// ---- DUTs/IO/PDOs/DO_X06_Pin4_Output_42CA91F7.TcDUT
{attribute 'GeneratedUsingTerminal: EP4378-1022-0017'}
{attribute addProperty BoxType "EP4378-1022-0017"}
{attribute addProperty Id "OutputAT %Q*BOOL1"}
{attribute addProperty CRC "1120571895"}
{attribute addProperty Size "1"}
TYPE DO_X06_Pin4_Output_42CA91F7 EXTENDS OutputBase_10CEE7DE :
STRUCT
	{attribute addProperty Name "Output"}
	Output AT %Q* : BOOL;
END_STRUCT
END_TYPE

// ---- DUTs/IO/PDOs/DO_X07_Pin4_Output_42CA91F7.TcDUT
{attribute 'GeneratedUsingTerminal: EP4378-1022-0017'}
{attribute addProperty BoxType "EP4378-1022-0017"}
{attribute addProperty Id "OutputAT %Q*BOOL1"}
{attribute addProperty CRC "1120571895"}
{attribute addProperty Size "1"}
TYPE DO_X07_Pin4_Output_42CA91F7 EXTENDS OutputBase_10CEE7DE :
STRUCT
	{attribute addProperty Name "Output"}
	Output AT %Q* : BOOL;
END_STRUCT
END_TYPE

// ---- DUTs/IO/PDOs/DO_X08_Pin4_Output_42CA91F7.TcDUT
{attribute 'GeneratedUsingTerminal: EP4378-1022-0017'}
{attribute addProperty BoxType "EP4378-1022-0017"}
{attribute addProperty Id "OutputAT %Q*BOOL1"}
{attribute addProperty CRC "1120571895"}
{attribute addProperty Size "1"}
TYPE DO_X08_Pin4_Output_42CA91F7 EXTENDS OutputBase_10CEE7DE :
STRUCT
	{attribute addProperty Name "Output"}
	Output AT %Q* : BOOL;
END_STRUCT
END_TYPE

// ---- DUTs/IO/PDOs/SSI_Inputs_0E3D8E33.TcDUT
{attribute 'GeneratedUsingTerminal: EP5001-0002-0016'}
{attribute addProperty BoxType "EP5001-0002-0016"}
{attribute addProperty Id "StatusAT %I*Status_ACC8459F6Counter_valueAT %I*UDINT4"}
{attribute addProperty CRC "238915123"}
{attribute addProperty Size "10"}
TYPE SSI_Inputs_0E3D8E33 EXTENDS InputBase_8311D824 :
STRUCT
	{attribute addProperty Name "Status"}
	Status AT %I* : Status_ACC8459F;
	{attribute addProperty Name "Counter_value"}
	Counter_value AT %I* : UDINT;
END_STRUCT
END_TYPE

// ---- DUTs/IO/PDOs/ENC_Status_compact_F4F89583.TcDUT
{attribute 'GeneratedUsingTerminal: EP5101-0002-0016'}
{attribute addProperty BoxType "EP5101-0002-0016"}
{attribute addProperty Id "StatusAT %I*Status_3A9E406C12Counter_valueAT %I*UINT2Latch_valueAT %I*UINT2"}
{attribute addProperty CRC "4109931907"}
{attribute addProperty Size "16"}
TYPE ENC_Status_compact_F4F89583 EXTENDS InputBase_8311D824 :
STRUCT
	{attribute addProperty Name "Status"}
	Status AT %I* : Status_3A9E406C;
	{attribute addProperty Name "Counter_value"}
	Counter_value AT %I* : UINT;
	{attribute addProperty Name "Latch_value"}
	Latch_value AT %I* : UINT;
END_STRUCT
END_TYPE

// ---- DUTs/IO/PDOs/ENC_Control_compact_E6DC9B25.TcDUT
{attribute 'GeneratedUsingTerminal: EP5101-0002-0016'}
{attribute addProperty BoxType "EP5101-0002-0016"}
{attribute addProperty Id "ControlAT %Q*Control_D500AB792Set_counter_valueAT %Q*UINT2"}
{attribute addProperty CRC "3873217317"}
{attribute addProperty Size "4"}
TYPE ENC_Control_compact_E6DC9B25 EXTENDS OutputBase_10CEE7DE :
STRUCT
	{attribute addProperty Name "Control"}
	Control AT %Q* : Control_D500AB79;
	{attribute addProperty Name "Set_counter_value"}
	Set_counter_value AT %Q* : UINT;
END_STRUCT
END_TYPE

// ---- DUTs/IO/PDOs/ENC_Status_compact_7D3464F3.TcDUT
{attribute 'GeneratedUsingTerminal: EP5101-0011-0016'}
{attribute addProperty BoxType "EP5101-0011-0016"}
{attribute addProperty Id "StatusAT %I*Status_D8D782C316Counter_valueAT %I*UINT2Latch_valueAT %I*UINT2"}
{attribute addProperty CRC "2100585715"}
{attribute addProperty Size "20"}
TYPE ENC_Status_compact_7D3464F3 EXTENDS InputBase_8311D824 :
STRUCT
	{attribute addProperty Name "Status"}
	Status AT %I* : Status_D8D782C3;
	{attribute addProperty Name "Counter_value"}
	Counter_value AT %I* : UINT;
	{attribute addProperty Name "Latch_value"}
	Latch_value AT %I* : UINT;
END_STRUCT
END_TYPE

// ---- DUTs/IO/PDOs/ENC_Control_compact_21E2D14D.TcDUT
{attribute 'GeneratedUsingTerminal: EP5101-0011-0016'}
{attribute addProperty BoxType "EP5101-0011-0016"}
{attribute addProperty Id "ControlAT %Q*Control_6EF2C5D04Set_counter_valueAT %Q*UINT2"}
{attribute addProperty CRC "568512845"}
{attribute addProperty Size "6"}
TYPE ENC_Control_compact_21E2D14D EXTENDS OutputBase_10CEE7DE :
STRUCT
	{attribute addProperty Name "Control"}
	Control AT %Q* : Control_6EF2C5D0;
	{attribute addProperty Name "Set_counter_value"}
	Set_counter_value AT %Q* : UINT;
END_STRUCT
END_TYPE

// ---- DUTs/IO/PDOs/ENC_Status_compact_4198EF3B.TcDUT
{attribute 'GeneratedUsingTerminal: EP5101-2011-0016'}
{attribute addProperty BoxType "EP5101-2011-0016"}
{attribute addProperty Id "StatusAT %I*Status_E2E79E8513Counter_valueAT %I*UINT2Latch_valueAT %I*UINT2"}
{attribute addProperty CRC "1100541755"}
{attribute addProperty Size "17"}
TYPE ENC_Status_compact_4198EF3B EXTENDS InputBase_8311D824 :
STRUCT
	{attribute addProperty Name "Status"}
	Status AT %I* : Status_E2E79E85;
	{attribute addProperty Name "Counter_value"}
	Counter_value AT %I* : UINT;
	{attribute addProperty Name "Latch_value"}
	Latch_value AT %I* : UINT;
END_STRUCT
END_TYPE

// ---- DUTs/IO/PDOs/COM_Inputs_6C2FC202.TcDUT
{attribute 'GeneratedUsingTerminal: EP6001-0002-0020'}
{attribute addProperty BoxType "EP6001-0002-0020"}
{attribute addProperty Id "StatusAT %I*UINT2Data_InAT %I*ARRAY[0..21] OF USINT22"}
{attribute addProperty CRC "1367962124"}
{attribute addProperty Size "24"}
TYPE COM_Inputs_6C2FC202 EXTENDS InputBase_8311D824 :
STRUCT
	{attribute addProperty Name "Status"}
	Status AT %I* : UINT;
	{attribute addProperty Name "Data_In"}
	Data_In AT %I* : ARRAY[0..21] OF USINT;
END_STRUCT
END_TYPE

// ---- DUTs/IO/PDOs/COM_Outputs_5D00B5E7.TcDUT
{attribute 'GeneratedUsingTerminal: EP6001-0002-0020'}
{attribute addProperty BoxType "EP6001-0002-0020"}
{attribute addProperty Id "CtrlAT %Q*UINT2Data_OutAT %Q*ARRAY[0..21] OF USINT22"}
{attribute addProperty CRC "875731620"}
{attribute addProperty Size "24"}
TYPE COM_Outputs_5D00B5E7 EXTENDS OutputBase_10CEE7DE :
STRUCT
	{attribute addProperty Name "Ctrl"}
	Ctrl AT %Q* : UINT;
	{attribute addProperty Name "Data_Out"}
	Data_Out AT %Q* : ARRAY[0..21] OF USINT;
END_STRUCT
END_TYPE

// ---- DUTs/IO/PDOs/COM_Inputs_Channel_C252EAC2.TcDUT
{attribute 'GeneratedUsingTerminal: EP6002-0002-0016'}
{attribute addProperty BoxType "EP6002-0002-0016"}
{attribute addProperty Id "StatusAT %I*WORD2Data_InAT %I*ARRAY[0..21] OF USINT22"}
{attribute addProperty CRC "3532970676"}
{attribute addProperty Size "24"}
TYPE COM_Inputs_Channel_C252EAC2 EXTENDS InputBase_8311D824 :
STRUCT
	{attribute addProperty Name "Status"}
	Status AT %I* : WORD;
	{attribute addProperty Name "Data_In"}
	Data_In AT %I* : ARRAY[0..21] OF USINT;
END_STRUCT
END_TYPE

// ---- DUTs/IO/PDOs/COM_Outputs_Channel_B336F4EE.TcDUT
{attribute 'GeneratedUsingTerminal: EP6002-0002-0016'}
{attribute addProperty BoxType "EP6002-0002-0016"}
{attribute addProperty Id "CtrlAT %Q*WORD2Data_OutAT %Q*ARRAY[0..21] OF USINT22"}
{attribute addProperty CRC "1305863315"}
{attribute addProperty Size "24"}
TYPE COM_Outputs_Channel_B336F4EE EXTENDS OutputBase_10CEE7DE :
STRUCT
	{attribute addProperty Name "Ctrl"}
	Ctrl AT %Q* : WORD;
	{attribute addProperty Name "Data_Out"}
	Data_Out AT %Q* : ARRAY[0..21] OF USINT;
END_STRUCT
END_TYPE

// ---- DUTs/IO/PDOs/COM_TxPDO_Map_Inputs_Channel_C252EAC2.TcDUT
{attribute 'GeneratedUsingTerminal: EP6002-0002-0017'}
{attribute addProperty BoxType "EP6002-0002-0017"}
{attribute addProperty Id "StatusAT %I*WORD2Data_InAT %I*ARRAY[0..21] OF USINT22"}
{attribute addProperty CRC "3532970676"}
{attribute addProperty Size "24"}
TYPE COM_TxPDO_Map_Inputs_Channel_C252EAC2 EXTENDS InputBase_8311D824 :
STRUCT
	{attribute addProperty Name "Status"}
	Status AT %I* : WORD;
	{attribute addProperty Name "Data_In"}
	Data_In AT %I* : ARRAY[0..21] OF USINT;
END_STRUCT
END_TYPE

// ---- DUTs/IO/PDOs/COM_RxPDO_Map_Outputs_Channel_B336F4EE.TcDUT
{attribute 'GeneratedUsingTerminal: EP6002-0002-0017'}
{attribute addProperty BoxType "EP6002-0002-0017"}
{attribute addProperty Id "CtrlAT %Q*WORD2Data_OutAT %Q*ARRAY[0..21] OF USINT22"}
{attribute addProperty CRC "1305863315"}
{attribute addProperty Size "24"}
TYPE COM_RxPDO_Map_Outputs_Channel_B336F4EE EXTENDS OutputBase_10CEE7DE :
STRUCT
	{attribute addProperty Name "Ctrl"}
	Ctrl AT %Q* : WORD;
	{attribute addProperty Name "Data_Out"}
	Data_Out AT %Q* : ARRAY[0..21] OF USINT;
END_STRUCT
END_TYPE

// ---- DUTs/IO/PDOs/COM_TxPDO_Map_Inputs_Channel_6C2FC202.TcDUT
{attribute 'GeneratedUsingTerminal: EP6002-0002-0023'}
{attribute addProperty BoxType "EP6002-0002-0023"}
{attribute addProperty Id "StatusAT %I*UINT2Data_InAT %I*ARRAY[0..21] OF USINT22"}
{attribute addProperty CRC "1367962124"}
{attribute addProperty Size "24"}
TYPE COM_TxPDO_Map_Inputs_Channel_6C2FC202 EXTENDS InputBase_8311D824 :
STRUCT
	{attribute addProperty Name "Status"}
	Status AT %I* : UINT;
	{attribute addProperty Name "Data_In"}
	Data_In AT %I* : ARRAY[0..21] OF USINT;
END_STRUCT
END_TYPE

// ---- DUTs/IO/PDOs/COM_RxPDO_Map_Outputs_Channel_5D00B5E7.TcDUT
{attribute 'GeneratedUsingTerminal: EP6002-0002-0023'}
{attribute addProperty BoxType "EP6002-0002-0023"}
{attribute addProperty Id "CtrlAT %Q*UINT2Data_OutAT %Q*ARRAY[0..21] OF USINT22"}
{attribute addProperty CRC "875731620"}
{attribute addProperty Size "24"}
TYPE COM_RxPDO_Map_Outputs_Channel_5D00B5E7 EXTENDS OutputBase_10CEE7DE :
STRUCT
	{attribute addProperty Name "Ctrl"}
	Ctrl AT %Q* : UINT;
	{attribute addProperty Name "Data_Out"}
	Data_Out AT %Q* : ARRAY[0..21] OF USINT;
END_STRUCT
END_TYPE

// ---- DUTs/IO/PDOs/DIS_Inputs_E0E384E3.TcDUT
{attribute 'GeneratedUsingTerminal: EP6090-0000-0017'}
{attribute addProperty BoxType "EP6090-0000-0017"}
{attribute addProperty Id "StatusAT %I*Status_E3E7FD126"}
{attribute addProperty CRC "3773007075"}
{attribute addProperty Size "6"}
TYPE DIS_Inputs_E0E384E3 EXTENDS InputBase_8311D824 :
STRUCT
	{attribute addProperty Name "Status"}
	Status AT %I* : Status_E3E7FD12;
END_STRUCT
END_TYPE

// ---- DUTs/IO/PDOs/DIS_Outputs_6C9BFFEE.TcDUT
{attribute 'GeneratedUsingTerminal: EP6090-0000-0017'}
{attribute addProperty BoxType "EP6090-0000-0017"}
{attribute addProperty Id "Value_rowAT %Q*ARRAY[0..1] OF INT4"}
{attribute addProperty CRC "4003442326"}
{attribute addProperty Size "4"}
TYPE DIS_Outputs_6C9BFFEE EXTENDS OutputBase_10CEE7DE :
STRUCT
	{attribute addProperty Name "Value_row"}
	Value_row AT %Q* : ARRAY[0..1] OF INT;
END_STRUCT
END_TYPE

// ---- DUTs/IO/PDOs/DeviceState_Inputs_Device_A1210598.TcDUT
{attribute 'GeneratedUsingTerminal: EP6224-0002-0016'}
{attribute addProperty BoxType "EP6224-0002-0016"}
{attribute addProperty Id "Device_DiagAT %I*BOOL1Device_StateAT %I*BOOL1"}
{attribute addProperty CRC "2703295896"}
{attribute addProperty Size "2"}
TYPE DeviceState_Inputs_Device_A1210598 EXTENDS InputBase_8311D824 :
STRUCT
	{attribute addProperty Name "Device_Diag"}
	Device_Diag AT %I* : BOOL;
	{attribute addProperty Name "Device_State"}
	Device_State AT %I* : BOOL;
END_STRUCT
END_TYPE

// ---- DUTs/IO/PDOs/DeviceState_Inputs_4751FF76.TcDUT
{attribute 'GeneratedUsingTerminal: EP6224-0002-0016'}
{attribute addProperty BoxType "EP6224-0002-0016"}
{attribute addProperty Id "State_Ch1AT %I*USINT1State_Ch2AT %I*USINT1State_Ch3AT %I*USINT1State_Ch4AT %I*USINT1"}
{attribute addProperty CRC "1196556150"}
{attribute addProperty Size "4"}
TYPE DeviceState_Inputs_4751FF76 EXTENDS InputBase_8311D824 :
STRUCT
	{attribute addProperty Name "State_Ch1"}
	State_Ch1 AT %I* : USINT;
	{attribute addProperty Name "State_Ch2"}
	State_Ch2 AT %I* : USINT;
	{attribute addProperty Name "State_Ch3"}
	State_Ch3 AT %I* : USINT;
	{attribute addProperty Name "State_Ch4"}
	State_Ch4 AT %I* : USINT;
END_STRUCT
END_TYPE

// ---- DUTs/IO/PDOs/Digital_Inputs_FE042239.TcDUT
{attribute 'GeneratedUsingTerminal: EP6224-0002-0016'}
{attribute addProperty BoxType "EP6224-0002-0016"}
{attribute addProperty Id "DI_X01_Pin2AT %I*BOOL1DI_X02_Pin2AT %I*BOOL1DI_X03_Pin2AT %I*BOOL1DI_X04_Pin2AT %I*BOOL1"}
{attribute addProperty CRC "4261683769"}
{attribute addProperty Size "4"}
TYPE Digital_Inputs_FE042239 EXTENDS InputBase_8311D824 :
STRUCT
	{attribute addProperty Name "DI_X01_Pin2"}
	DI_X01_Pin2 AT %I* : BOOL;
	{attribute addProperty Name "DI_X02_Pin2"}
	DI_X02_Pin2 AT %I* : BOOL;
	{attribute addProperty Name "DI_X03_Pin2"}
	DI_X03_Pin2 AT %I* : BOOL;
	{attribute addProperty Name "DI_X04_Pin2"}
	DI_X04_Pin2 AT %I* : BOOL;
END_STRUCT
END_TYPE

// ---- DUTs/IO/PDOs/InfoData_90184F0C.TcDUT
{attribute 'GeneratedUsingTerminal: EP6224-0002-0016'}
{attribute addProperty BoxType "EP6224-0002-0016"}
{attribute addProperty Id "AdsAddrAT %I*AMSADDR8AoeNetIdAT %I*AMSNETID6StateAT %I*UINT2"}
{attribute addProperty CRC "2417512204"}
{attribute addProperty Size "16"}
TYPE InfoData_90184F0C EXTENDS InputBase_8311D824 :
STRUCT
	{attribute addProperty Name "AdsAddr"}
	AdsAddr AT %I* : AMSADDR;
	{attribute addProperty Name "AoeNetId"}
	AoeNetId AT %I* : AMSNETID;
	{attribute addProperty Name "State"}
	State AT %I* : UINT;
END_STRUCT
END_TYPE

// ---- DUTs/IO/PDOs/Module_1_DeviceState_Inputs_Device_5322301C.TcDUT
{attribute 'GeneratedUsingTerminal: EP6224-0002-0016'}
{attribute addProperty BoxType "EP6224-0002-0016"}
{attribute addProperty Id "DeviceState_Inputs_DeviceDeviceState_Inputs_Device_A12105982"}
{attribute addProperty CRC "1394749468"}
{attribute addProperty Size "2"}
TYPE Module_1_DeviceState_Inputs_Device_5322301C :
STRUCT
	{attribute addProperty Name "DeviceState_Inputs_Device"}
	DeviceState_Inputs_Device  : DeviceState_Inputs_Device_A1210598;
END_STRUCT
END_TYPE

// ---- DUTs/IO/PDOs/Module_2_DeviceState_Inputs_BD6C7035.TcDUT
{attribute 'GeneratedUsingTerminal: EP6224-0002-0016'}
{attribute addProperty BoxType "EP6224-0002-0016"}
{attribute addProperty Id "DeviceState_InputsDeviceState_Inputs_4751FF764"}
{attribute addProperty CRC "3178000437"}
{attribute addProperty Size "4"}
TYPE Module_2_DeviceState_Inputs_BD6C7035 :
STRUCT
	{attribute addProperty Name "DeviceState_Inputs"}
	DeviceState_Inputs  : DeviceState_Inputs_4751FF76;
END_STRUCT
END_TYPE

// ---- DUTs/IO/PDOs/Module_7_Digital_Inputs_F29732B3.TcDUT
{attribute 'GeneratedUsingTerminal: EP6224-0002-0016'}
{attribute addProperty BoxType "EP6224-0002-0016"}
{attribute addProperty Id "Digital_InputsDigital_Inputs_FE0422394"}
{attribute addProperty CRC "4069995187"}
{attribute addProperty Size "4"}
TYPE Module_7_Digital_Inputs_F29732B3 :
STRUCT
	{attribute addProperty Name "Digital_Inputs"}
	Digital_Inputs  : Digital_Inputs_FE042239;
END_STRUCT
END_TYPE

// ---- DUTs/IO/PDOs/Digital_Inputs_8749E151.TcDUT
{attribute 'GeneratedUsingTerminal: EP6224-0042-0016'}
{attribute addProperty BoxType "EP6224-0042-0016"}
{attribute addProperty Id "DI_X01_Pin2AT %I*BOOL1DI_X01_Pin4AT %I*BOOL1DI_X02_Pin2AT %I*BOOL1DI_X02_Pin4AT %I*BOOL1DI_X05_Pin2AT %I*BOOL1DI_X05_Pin4AT %I*BOOL1DI_X06_Pin2AT %I*BOOL1DI_X06_Pin4AT %I*BOOL1"}
{attribute addProperty CRC "2269765969"}
{attribute addProperty Size "8"}
TYPE Digital_Inputs_8749E151 EXTENDS InputBase_8311D824 :
STRUCT
	{attribute addProperty Name "DI_X01_Pin2"}
	DI_X01_Pin2 AT %I* : BOOL;
	{attribute addProperty Name "DI_X01_Pin4"}
	DI_X01_Pin4 AT %I* : BOOL;
	{attribute addProperty Name "DI_X02_Pin2"}
	DI_X02_Pin2 AT %I* : BOOL;
	{attribute addProperty Name "DI_X02_Pin4"}
	DI_X02_Pin4 AT %I* : BOOL;
	{attribute addProperty Name "DI_X05_Pin2"}
	DI_X05_Pin2 AT %I* : BOOL;
	{attribute addProperty Name "DI_X05_Pin4"}
	DI_X05_Pin4 AT %I* : BOOL;
	{attribute addProperty Name "DI_X06_Pin2"}
	DI_X06_Pin2 AT %I* : BOOL;
	{attribute addProperty Name "DI_X06_Pin4"}
	DI_X06_Pin4 AT %I* : BOOL;
END_STRUCT
END_TYPE

// ---- DUTs/IO/PDOs/Module_7_Digital_Inputs_DAAE149B.TcDUT
{attribute 'GeneratedUsingTerminal: EP6224-0042-0016'}
{attribute addProperty BoxType "EP6224-0042-0016"}
{attribute addProperty Id "Digital_InputsDigital_Inputs_8749E1518"}
{attribute addProperty CRC "3668841627"}
{attribute addProperty Size "8"}
TYPE Module_7_Digital_Inputs_DAAE149B :
STRUCT
	{attribute addProperty Name "Digital_Inputs"}
	Digital_Inputs  : Digital_Inputs_8749E151;
END_STRUCT
END_TYPE

// ---- DUTs/IO/PDOs/EMPTY_STRUCTURE.TcDUT
{attribute 'GeneratedUsingTerminal: EP6224-2022-0016'}
{attribute addProperty BoxType "EP6224-2022-0016"}
{attribute addProperty Id "EMPTY_STRUCTURE"}
{attribute addProperty CRC "0"}
{attribute addProperty Size "0"}
TYPE EMPTY_STRUCTURE :
STRUCT
END_STRUCT
END_TYPE

// ---- DUTs/IO/PDOs/DeviceState_Inputs_C7251DC9.TcDUT
{attribute 'GeneratedUsingTerminal: EP6228-0022-0016'}
{attribute addProperty BoxType "EP6228-0022-0016"}
{attribute addProperty Id "State_Ch1AT %I*USINT1State_Ch2AT %I*USINT1State_Ch3AT %I*USINT1State_Ch4AT %I*USINT1State_Ch5AT %I*USINT1State_Ch6AT %I*USINT1State_Ch7AT %I*USINT1State_Ch8AT %I*USINT1"}
{attribute addProperty CRC "3341098441"}
{attribute addProperty Size "8"}
TYPE DeviceState_Inputs_C7251DC9 EXTENDS InputBase_8311D824 :
STRUCT
	{attribute addProperty Name "State_Ch1"}
	State_Ch1 AT %I* : USINT;
	{attribute addProperty Name "State_Ch2"}
	State_Ch2 AT %I* : USINT;
	{attribute addProperty Name "State_Ch3"}
	State_Ch3 AT %I* : USINT;
	{attribute addProperty Name "State_Ch4"}
	State_Ch4 AT %I* : USINT;
	{attribute addProperty Name "State_Ch5"}
	State_Ch5 AT %I* : USINT;
	{attribute addProperty Name "State_Ch6"}
	State_Ch6 AT %I* : USINT;
	{attribute addProperty Name "State_Ch7"}
	State_Ch7 AT %I* : USINT;
	{attribute addProperty Name "State_Ch8"}
	State_Ch8 AT %I* : USINT;
END_STRUCT
END_TYPE

// ---- DUTs/IO/PDOs/Module_2_DeviceState_Inputs_B92A0D6A.TcDUT
{attribute 'GeneratedUsingTerminal: EP6228-0022-0016'}
{attribute addProperty BoxType "EP6228-0022-0016"}
{attribute addProperty Id "DeviceState_InputsDeviceState_Inputs_C7251DC98"}
{attribute addProperty CRC "3106540906"}
{attribute addProperty Size "8"}
TYPE Module_2_DeviceState_Inputs_B92A0D6A :
STRUCT
	{attribute addProperty Name "DeviceState_Inputs"}
	DeviceState_Inputs  : DeviceState_Inputs_C7251DC9;
END_STRUCT
END_TYPE

// ---- DUTs/IO/PDOs/Digital_Inputs_83D7E782.TcDUT
{attribute 'GeneratedUsingTerminal: EP6228-0042-0016'}
{attribute addProperty BoxType "EP6228-0042-0016"}
{attribute addProperty Id "Pin2_Ch1AT %I*BOOL1Pin2_Ch2AT %I*BOOL1Pin2_Ch3AT %I*BOOL1Pin2_Ch4AT %I*BOOL1Pin2_Ch5AT %I*BOOL1Pin2_Ch6AT %I*BOOL1Pin2_Ch7AT %I*BOOL1Pin2_Ch8AT %I*BOOL1"}
{attribute addProperty CRC "2211964802"}
{attribute addProperty Size "8"}
TYPE Digital_Inputs_83D7E782 EXTENDS InputBase_8311D824 :
STRUCT
	{attribute addProperty Name "Pin2_Ch1"}
	Pin2_Ch1 AT %I* : BOOL;
	{attribute addProperty Name "Pin2_Ch2"}
	Pin2_Ch2 AT %I* : BOOL;
	{attribute addProperty Name "Pin2_Ch3"}
	Pin2_Ch3 AT %I* : BOOL;
	{attribute addProperty Name "Pin2_Ch4"}
	Pin2_Ch4 AT %I* : BOOL;
	{attribute addProperty Name "Pin2_Ch5"}
	Pin2_Ch5 AT %I* : BOOL;
	{attribute addProperty Name "Pin2_Ch6"}
	Pin2_Ch6 AT %I* : BOOL;
	{attribute addProperty Name "Pin2_Ch7"}
	Pin2_Ch7 AT %I* : BOOL;
	{attribute addProperty Name "Pin2_Ch8"}
	Pin2_Ch8 AT %I* : BOOL;
END_STRUCT
END_TYPE

// ---- DUTs/IO/PDOs/Module_11_Digital_Inputs_33FD8372.TcDUT
{attribute 'GeneratedUsingTerminal: EP6228-0042-0016'}
{attribute addProperty BoxType "EP6228-0042-0016"}
{attribute addProperty Id "Digital_InputsDigital_Inputs_83D7E7828"}
{attribute addProperty CRC "872252274"}
{attribute addProperty Size "8"}
TYPE Module_11_Digital_Inputs_33FD8372 :
STRUCT
	{attribute addProperty Name "Digital_Inputs"}
	Digital_Inputs  : Digital_Inputs_83D7E782;
END_STRUCT
END_TYPE

// ---- DUTs/IO/PDOs/Digital_Inputs_3DEC2D27.TcDUT
{attribute 'GeneratedUsingTerminal: EP6228-3132-0016'}
{attribute addProperty BoxType "EP6228-3132-0016"}
{attribute addProperty Id "Pin2_Ch1AT %I*BOOL1Pin2_Ch2AT %I*BOOL1Pin2_Ch5AT %I*BOOL1Pin2_Ch6AT %I*BOOL1"}
{attribute addProperty CRC "1038888231"}
{attribute addProperty Size "4"}
TYPE Digital_Inputs_3DEC2D27 EXTENDS InputBase_8311D824 :
STRUCT
	{attribute addProperty Name "Pin2_Ch1"}
	Pin2_Ch1 AT %I* : BOOL;
	{attribute addProperty Name "Pin2_Ch2"}
	Pin2_Ch2 AT %I* : BOOL;
	{attribute addProperty Name "Pin2_Ch5"}
	Pin2_Ch5 AT %I* : BOOL;
	{attribute addProperty Name "Pin2_Ch6"}
	Pin2_Ch6 AT %I* : BOOL;
END_STRUCT
END_TYPE

// ---- DUTs/IO/PDOs/Module_11_Digital_Inputs_36A01C39.TcDUT
{attribute 'GeneratedUsingTerminal: EP6228-3132-0016'}
{attribute addProperty BoxType "EP6228-3132-0016"}
{attribute addProperty Id "Digital_InputsDigital_Inputs_3DEC2D274"}
{attribute addProperty CRC "916462649"}
{attribute addProperty Size "4"}
TYPE Module_11_Digital_Inputs_36A01C39 :
STRUCT
	{attribute addProperty Name "Digital_Inputs"}
	Digital_Inputs  : Digital_Inputs_3DEC2D27;
END_STRUCT
END_TYPE

// ---- DUTs/IO/PDOs/ENC_Status_compact_4D066E1A.TcDUT
{attribute 'GeneratedUsingTerminal: EP7041-0002-0016'}
{attribute addProperty BoxType "EP7041-0002-0016"}
{attribute addProperty Id "StatusAT %I*Status_8CBE219F12Counter_valueAT %I*UINT2Latch_valueAT %I*UINT2"}
{attribute addProperty CRC "1292267034"}
{attribute addProperty Size "16"}
TYPE ENC_Status_compact_4D066E1A EXTENDS InputBase_8311D824 :
STRUCT
	{attribute addProperty Name "Status"}
	Status AT %I* : Status_8CBE219F;
	{attribute addProperty Name "Counter_value"}
	Counter_value AT %I* : UINT;
	{attribute addProperty Name "Latch_value"}
	Latch_value AT %I* : UINT;
END_STRUCT
END_TYPE

// ---- DUTs/IO/PDOs/STM_Status_36ED096F.TcDUT
{attribute 'GeneratedUsingTerminal: EP7041-0002-0016'}
{attribute addProperty BoxType "EP7041-0002-0016"}
{attribute addProperty Id "StatusAT %I*Status_B679584511"}
{attribute addProperty CRC "921504111"}
{attribute addProperty Size "11"}
TYPE STM_Status_36ED096F EXTENDS InputBase_8311D824 :
STRUCT
	{attribute addProperty Name "Status"}
	Status AT %I* : Status_B6795845;
END_STRUCT
END_TYPE

// ---- DUTs/IO/PDOs/STM_Control_BA4CE352.TcDUT
{attribute 'GeneratedUsingTerminal: EP7041-0002-0016'}
{attribute addProperty BoxType "EP7041-0002-0016"}
{attribute addProperty Id "ControlAT %Q*Control_5FD4673D4"}
{attribute addProperty CRC "3125601106"}
{attribute addProperty Size "4"}
TYPE STM_Control_BA4CE352 EXTENDS OutputBase_10CEE7DE :
STRUCT
	{attribute addProperty Name "Control"}
	Control AT %Q* : Control_5FD4673D;
END_STRUCT
END_TYPE

// ---- DUTs/IO/PDOs/STM_Velocity_A47A3F41.TcDUT
{attribute 'GeneratedUsingTerminal: EP7041-0002-0016'}
{attribute addProperty BoxType "EP7041-0002-0016"}
{attribute addProperty Id "VelocityAT %Q*INT2"}
{attribute addProperty CRC "2759475009"}
{attribute addProperty Size "2"}
TYPE STM_Velocity_A47A3F41 EXTENDS OutputBase_10CEE7DE :
STRUCT
	{attribute addProperty Name "Velocity"}
	Velocity AT %Q* : INT;
END_STRUCT
END_TYPE

// ---- DUTs/IO/PDOs/InfoData_8DF4E0C5.TcDUT
{attribute 'GeneratedUsingTerminal: EP7041-0002-0016'}
{attribute addProperty BoxType "EP7041-0002-0016"}
{attribute addProperty Id "AdsAddrAT %I*AMSADDR8Chn0AT %I*USINT1StateAT %I*UINT2"}
{attribute addProperty CRC "2381635781"}
{attribute addProperty Size "11"}
TYPE InfoData_8DF4E0C5 EXTENDS InputBase_8311D824 :
STRUCT
	{attribute addProperty Name "AdsAddr"}
	AdsAddr AT %I* : AMSADDR;
	{attribute addProperty Name "Chn0"}
	Chn0 AT %I* : USINT;
	{attribute addProperty Name "State"}
	State AT %I* : UINT;
END_STRUCT
END_TYPE

// ---- DUTs/IO/PDOs/InfoData_6538CF5F.TcDUT
{attribute 'GeneratedUsingTerminal: EP7041-0002-0018'}
{attribute addProperty BoxType "EP7041-0002-0018"}
{attribute addProperty Id "AdsAddrAT %I*AMSADDR8Chn0AT %I*USINT1Chn1AT %I*USINT1StateAT %I*UINT2"}
{attribute addProperty CRC "1698221919"}
{attribute addProperty Size "12"}
TYPE InfoData_6538CF5F EXTENDS InputBase_8311D824 :
STRUCT
	{attribute addProperty Name "AdsAddr"}
	AdsAddr AT %I* : AMSADDR;
	{attribute addProperty Name "Chn0"}
	Chn0 AT %I* : USINT;
	{attribute addProperty Name "Chn1"}
	Chn1 AT %I* : USINT;
	{attribute addProperty Name "State"}
	State AT %I* : UINT;
END_STRUCT
END_TYPE

// ---- DUTs/IO/PDOs/STM_Status_DE0D6B37.TcDUT
{attribute 'GeneratedUsingTerminal: EP7041-3002-0016'}
{attribute addProperty BoxType "EP7041-3002-0016"}
{attribute addProperty Id "StatusAT %I*Status_1E008DB912"}
{attribute addProperty CRC "3725421367"}
{attribute addProperty Size "12"}
TYPE STM_Status_DE0D6B37 EXTENDS InputBase_8311D824 :
STRUCT
	{attribute addProperty Name "Status"}
	Status AT %I* : Status_1E008DB9;
END_STRUCT
END_TYPE

// ---- DUTs/IO/PDOs/FB_Position_3FA094ED.TcDUT
{attribute 'GeneratedUsingTerminal: EP7211-0034-0029'}
{attribute addProperty BoxType "EP7211-0034-0029"}
{attribute addProperty Id "PositionAT %I*UDINT4"}
{attribute addProperty CRC "1067488493"}
{attribute addProperty Size "4"}
TYPE FB_Position_3FA094ED EXTENDS InputBase_8311D824 :
STRUCT
	{attribute addProperty Name "Position"}
	Position AT %I* : UDINT;
END_STRUCT
END_TYPE

// ---- DUTs/IO/PDOs/DRV_Statusword_9B36FDFC.TcDUT
{attribute 'GeneratedUsingTerminal: EP7211-0034-0029'}
{attribute addProperty BoxType "EP7211-0034-0029"}
{attribute addProperty Id "StatuswordAT %I*UINT2"}
{attribute addProperty CRC "2604072444"}
{attribute addProperty Size "2"}
TYPE DRV_Statusword_9B36FDFC EXTENDS InputBase_8311D824 :
STRUCT
	{attribute addProperty Name "Statusword"}
	Statusword AT %I* : UINT;
END_STRUCT
END_TYPE

// ---- DUTs/IO/PDOs/DRV_Controlword_F3F14721.TcDUT
{attribute 'GeneratedUsingTerminal: EP7211-0034-0029'}
{attribute addProperty BoxType "EP7211-0034-0029"}
{attribute addProperty Id "ControlwordAT %Q*UINT2"}
{attribute addProperty CRC "4092675873"}
{attribute addProperty Size "2"}
TYPE DRV_Controlword_F3F14721 EXTENDS OutputBase_10CEE7DE :
STRUCT
	{attribute addProperty Name "Controlword"}
	Controlword AT %Q* : UINT;
END_STRUCT
END_TYPE

// ---- DUTs/IO/PDOs/DRV_Target_velocity_08A9583B.TcDUT
{attribute 'GeneratedUsingTerminal: EP7211-0034-0029'}
{attribute addProperty BoxType "EP7211-0034-0029"}
{attribute addProperty Id "Target_velocityAT %Q*DINT4"}
{attribute addProperty CRC "145315899"}
{attribute addProperty Size "4"}
TYPE DRV_Target_velocity_08A9583B EXTENDS OutputBase_10CEE7DE :
STRUCT
	{attribute addProperty Name "Target_velocity"}
	Target_velocity AT %Q* : DINT;
END_STRUCT
END_TYPE

// ---- DUTs/IO/PDOs/InfoData_96C94FAE.TcDUT
{attribute 'GeneratedUsingTerminal: EP7211-0034-0029'}
{attribute addProperty BoxType "EP7211-0034-0029"}
{attribute addProperty Id "AdsAddrAT %I*AMSADDR8DcOutputShiftAT %I*DINT4DcInputShiftAT %I*DINT4Chn0AT %I*USINT1StateAT %I*UINT2"}
{attribute addProperty CRC "2529775534"}
{attribute addProperty Size "19"}
TYPE InfoData_96C94FAE EXTENDS InputBase_8311D824 :
STRUCT
	{attribute addProperty Name "AdsAddr"}
	AdsAddr AT %I* : AMSADDR;
	{attribute addProperty Name "DcOutputShift"}
	DcOutputShift AT %I* : DINT;
	{attribute addProperty Name "DcInputShift"}
	DcInputShift AT %I* : DINT;
	{attribute addProperty Name "Chn0"}
	Chn0 AT %I* : USINT;
	{attribute addProperty Name "State"}
	State AT %I* : UINT;
END_STRUCT
END_TYPE

// ---- DUTs/IO/PDOs/InfoData_6185D47C.TcDUT
{attribute 'GeneratedUsingTerminal: EP7211-0034-0030'}
{attribute addProperty BoxType "EP7211-0034-0030"}
{attribute addProperty Id "AdsAddrAT %I*AMSADDR8DcOutputShiftAT %I*DINT4DcInputShiftAT %I*DINT4Chn0AT %I*USINT1Chn1AT %I*USINT1StateAT %I*UINT2"}
{attribute addProperty CRC "1636160636"}
{attribute addProperty Size "20"}
TYPE InfoData_6185D47C EXTENDS InputBase_8311D824 :
STRUCT
	{attribute addProperty Name "AdsAddr"}
	AdsAddr AT %I* : AMSADDR;
	{attribute addProperty Name "DcOutputShift"}
	DcOutputShift AT %I* : DINT;
	{attribute addProperty Name "DcInputShift"}
	DcInputShift AT %I* : DINT;
	{attribute addProperty Name "Chn0"}
	Chn0 AT %I* : USINT;
	{attribute addProperty Name "Chn1"}
	Chn1 AT %I* : USINT;
	{attribute addProperty Name "State"}
	State AT %I* : UINT;
END_STRUCT
END_TYPE

// ---- DUTs/IO/PDOs/DS402_Statusword_9B36FDFC.TcDUT
{attribute 'GeneratedUsingTerminal: EP7211-0035-0029'}
{attribute addProperty BoxType "EP7211-0035-0029"}
{attribute addProperty Id "StatuswordAT %I*UINT2"}
{attribute addProperty CRC "2604072444"}
{attribute addProperty Size "2"}
TYPE DS402_Statusword_9B36FDFC EXTENDS InputBase_8311D824 :
STRUCT
	{attribute addProperty Name "Statusword"}
	Statusword AT %I* : UINT;
END_STRUCT
END_TYPE

// ---- DUTs/IO/PDOs/DS402_Position_actual_value_07DC4C74.TcDUT
{attribute 'GeneratedUsingTerminal: EP7211-0035-0029'}
{attribute addProperty BoxType "EP7211-0035-0029"}
{attribute addProperty Id "Position_actual_valueAT %I*UDINT4"}
{attribute addProperty CRC "131878004"}
{attribute addProperty Size "4"}
TYPE DS402_Position_actual_value_07DC4C74 EXTENDS InputBase_8311D824 :
STRUCT
	{attribute addProperty Name "Position_actual_value"}
	Position_actual_value AT %I* : UDINT;
END_STRUCT
END_TYPE

// ---- DUTs/IO/PDOs/DS402_Controlword_F3F14721.TcDUT
{attribute 'GeneratedUsingTerminal: EP7211-0035-0029'}
{attribute addProperty BoxType "EP7211-0035-0029"}
{attribute addProperty Id "ControlwordAT %Q*UINT2"}
{attribute addProperty CRC "4092675873"}
{attribute addProperty Size "2"}
TYPE DS402_Controlword_F3F14721 EXTENDS OutputBase_10CEE7DE :
STRUCT
	{attribute addProperty Name "Controlword"}
	Controlword AT %Q* : UINT;
END_STRUCT
END_TYPE

// ---- DUTs/IO/PDOs/DS402_Target_velocity_08A9583B.TcDUT
{attribute 'GeneratedUsingTerminal: EP7211-0035-0029'}
{attribute addProperty BoxType "EP7211-0035-0029"}
{attribute addProperty Id "Target_velocityAT %Q*DINT4"}
{attribute addProperty CRC "145315899"}
{attribute addProperty Size "4"}
TYPE DS402_Target_velocity_08A9583B EXTENDS OutputBase_10CEE7DE :
STRUCT
	{attribute addProperty Name "Target_velocity"}
	Target_velocity AT %Q* : DINT;
END_STRUCT
END_TYPE

// ---- DUTs/IO/PDOs/ENC_Status_compact_Channel_DC559AB0.TcDUT
{attribute 'GeneratedUsingTerminal: EP7342-0002-0016'}
{attribute addProperty BoxType "EP7342-0002-0016"}
{attribute addProperty Id "StatusAT %I*Status_3035BE2E10Counter_valueAT %I*UINT2Latch_valueAT %I*UINT2"}
{attribute addProperty CRC "3696597680"}
{attribute addProperty Size "14"}
TYPE ENC_Status_compact_Channel_DC559AB0 EXTENDS InputBase_8311D824 :
STRUCT
	{attribute addProperty Name "Status"}
	Status AT %I* : Status_3035BE2E;
	{attribute addProperty Name "Counter_value"}
	Counter_value AT %I* : UINT;
	{attribute addProperty Name "Latch_value"}
	Latch_value AT %I* : UINT;
END_STRUCT
END_TYPE

// ---- DUTs/IO/PDOs/DCM_Status_Channel_36ED096F.TcDUT
{attribute 'GeneratedUsingTerminal: EP7342-0002-0016'}
{attribute addProperty BoxType "EP7342-0002-0016"}
{attribute addProperty Id "StatusAT %I*Status_B679584511"}
{attribute addProperty CRC "921504111"}
{attribute addProperty Size "11"}
TYPE DCM_Status_Channel_36ED096F EXTENDS InputBase_8311D824 :
STRUCT
	{attribute addProperty Name "Status"}
	Status AT %I* : Status_B6795845;
END_STRUCT
END_TYPE

// ---- DUTs/IO/PDOs/ENC_Control_compact_Channel_2E82BC43.TcDUT
{attribute 'GeneratedUsingTerminal: EP7342-0002-0016'}
{attribute addProperty BoxType "EP7342-0002-0016"}
{attribute addProperty Id "ControlAT %Q*Control_F189B7373Set_counter_valueAT %Q*UINT2"}
{attribute addProperty CRC "780319811"}
{attribute addProperty Size "5"}
TYPE ENC_Control_compact_Channel_2E82BC43 EXTENDS OutputBase_10CEE7DE :
STRUCT
	{attribute addProperty Name "Control"}
	Control AT %Q* : Control_F189B737;
	{attribute addProperty Name "Set_counter_value"}
	Set_counter_value AT %Q* : UINT;
END_STRUCT
END_TYPE

// ---- DUTs/IO/PDOs/DCM_Control_Channel_5A8B5016.TcDUT
{attribute 'GeneratedUsingTerminal: EP7342-0002-0016'}
{attribute addProperty BoxType "EP7342-0002-0016"}
{attribute addProperty Id "ControlAT %Q*Control_C948E0F23"}
{attribute addProperty CRC "1519079446"}
{attribute addProperty Size "3"}
TYPE DCM_Control_Channel_5A8B5016 EXTENDS OutputBase_10CEE7DE :
STRUCT
	{attribute addProperty Name "Control"}
	Control AT %Q* : Control_C948E0F2;
END_STRUCT
END_TYPE

// ---- DUTs/IO/PDOs/DCM_Velocity_Channel_A47A3F41.TcDUT
{attribute 'GeneratedUsingTerminal: EP7342-0002-0016'}
{attribute addProperty BoxType "EP7342-0002-0016"}
{attribute addProperty Id "VelocityAT %Q*INT2"}
{attribute addProperty CRC "2759475009"}
{attribute addProperty Size "2"}
TYPE DCM_Velocity_Channel_A47A3F41 EXTENDS OutputBase_10CEE7DE :
STRUCT
	{attribute addProperty Name "Velocity"}
	Velocity AT %Q* : INT;
END_STRUCT
END_TYPE

// ---- DUTs/IO/PDOs/InfoData_939F71B6.TcDUT
{attribute 'GeneratedUsingTerminal: EP7342-0002-0016'}
{attribute addProperty BoxType "EP7342-0002-0016"}
{attribute addProperty Id "AdsAddrAT %I*AMSADDR8Chn0AT %I*USINT1Chn1AT %I*USINT1Chn2AT %I*USINT1Chn3AT %I*USINT1StateAT %I*UINT2"}
{attribute addProperty CRC "2476700086"}
{attribute addProperty Size "14"}
TYPE InfoData_939F71B6 EXTENDS InputBase_8311D824 :
STRUCT
	{attribute addProperty Name "AdsAddr"}
	AdsAddr AT %I* : AMSADDR;
	{attribute addProperty Name "Chn0"}
	Chn0 AT %I* : USINT;
	{attribute addProperty Name "Chn1"}
	Chn1 AT %I* : USINT;
	{attribute addProperty Name "Chn2"}
	Chn2 AT %I* : USINT;
	{attribute addProperty Name "Chn3"}
	Chn3 AT %I* : USINT;
	{attribute addProperty Name "State"}
	State AT %I* : UINT;
END_STRUCT
END_TYPE

// ---- DUTs/IO/PDOs/DI_Inputs_58955D1A.TcDUT
{attribute 'GeneratedUsingTerminal: EP7402-0057-0017'}
{attribute addProperty BoxType "EP7402-0057-0017"}
{attribute addProperty Id "InputAT %I*ARRAY[0..3] OF BOOL4Control_inputAT %I*ARRAY[0..3] OF BOOL4"}
{attribute addProperty CRC "56034484"}
{attribute addProperty Size "8"}
TYPE DI_Inputs_58955D1A EXTENDS InputBase_8311D824 :
STRUCT
	{attribute addProperty Name "Input"}
	Input AT %I* : ARRAY[0..3] OF BOOL;
	{attribute addProperty Name "Control_input"}
	Control_input AT %I* : ARRAY[0..3] OF BOOL;
END_STRUCT
END_TYPE

// ---- DUTs/IO/PDOs/STM_Status_Channel_99D1DFFA.TcDUT
{attribute 'GeneratedUsingTerminal: EP7402-0057-0017'}
{attribute addProperty BoxType "EP7402-0057-0017"}
{attribute addProperty Id "StatusAT %I*Status_725F98F27"}
{attribute addProperty CRC "2580668410"}
{attribute addProperty Size "7"}
TYPE STM_Status_Channel_99D1DFFA EXTENDS InputBase_8311D824 :
STRUCT
	{attribute addProperty Name "Status"}
	Status AT %I* : Status_725F98F2;
END_STRUCT
END_TYPE

// ---- DUTs/IO/PDOs/STM_Synchron_info_data_Channel_DD535D91.TcDUT
{attribute 'GeneratedUsingTerminal: EP7402-0057-0017'}
{attribute addProperty BoxType "EP7402-0057-0017"}
{attribute addProperty Id "Info_dataAT %I*ARRAY[0..2] OF UINT6"}
{attribute addProperty CRC "1532541242"}
{attribute addProperty Size "6"}
TYPE STM_Synchron_info_data_Channel_DD535D91 EXTENDS InputBase_8311D824 :
STRUCT
	{attribute addProperty Name "Info_data"}
	Info_data AT %I* : ARRAY[0..2] OF UINT;
END_STRUCT
END_TYPE

// ---- DUTs/IO/PDOs/STM_Inputs_Device_A41D8456.TcDUT
{attribute 'GeneratedUsingTerminal: EP7402-0057-0017'}
{attribute addProperty BoxType "EP7402-0057-0017"}
{attribute addProperty Id "Device_DiagAT %I*Device_Diag_1464ECF921"}
{attribute addProperty CRC "2753397846"}
{attribute addProperty Size "21"}
TYPE STM_Inputs_Device_A41D8456 EXTENDS InputBase_8311D824 :
STRUCT
	{attribute addProperty Name "Device_Diag"}
	Device_Diag AT %I* : Device_Diag_1464ECF9;
END_STRUCT
END_TYPE

// ---- DUTs/IO/PDOs/DO_Outputs_A241BD3A.TcDUT
{attribute 'GeneratedUsingTerminal: EP7402-0057-0017'}
{attribute addProperty BoxType "EP7402-0057-0017"}
{attribute addProperty Id "OutputAT %Q*ARRAY[0..3] OF BOOL4Control_outputAT %Q*ARRAY[0..3] OF BOOL4"}
{attribute addProperty CRC "905683247"}
{attribute addProperty Size "8"}
TYPE DO_Outputs_A241BD3A EXTENDS OutputBase_10CEE7DE :
STRUCT
	{attribute addProperty Name "Output"}
	Output AT %Q* : ARRAY[0..3] OF BOOL;
	{attribute addProperty Name "Control_output"}
	Control_output AT %Q* : ARRAY[0..3] OF BOOL;
END_STRUCT
END_TYPE

// ---- DUTs/IO/PDOs/STM_Control_Channel_F193EBCD.TcDUT
{attribute 'GeneratedUsingTerminal: EP7402-0057-0017'}
{attribute addProperty BoxType "EP7402-0057-0017"}
{attribute addProperty Id "ControlAT %Q*Control_F58A89C54"}
{attribute addProperty CRC "4053003213"}
{attribute addProperty Size "4"}
TYPE STM_Control_Channel_F193EBCD EXTENDS OutputBase_10CEE7DE :
STRUCT
	{attribute addProperty Name "Control"}
	Control AT %Q* : Control_F58A89C5;
END_STRUCT
END_TYPE

// ---- DUTs/IO/PDOs/STM_Target_Velocity_Channel_E69D8325.TcDUT
{attribute 'GeneratedUsingTerminal: EP7402-0057-0017'}
{attribute addProperty BoxType "EP7402-0057-0017"}
{attribute addProperty Id "VelocityAT %Q*INT2AccellerationAT %Q*UINT2DeccelerationAT %Q*UINT2"}
{attribute addProperty CRC "3869082405"}
{attribute addProperty Size "6"}
TYPE STM_Target_Velocity_Channel_E69D8325 EXTENDS OutputBase_10CEE7DE :
STRUCT
	{attribute addProperty Name "Velocity"}
	Velocity AT %Q* : INT;
	{attribute addProperty Name "Accelleration"}
	Accelleration AT %Q* : UINT;
	{attribute addProperty Name "Decceleration"}
	Decceleration AT %Q* : UINT;
END_STRUCT
END_TYPE

// ---- DUTs/IO/PDOs/TACHO_Single_Shaft_Mode_Input_Channel_C331CA3E.TcDUT
{attribute 'GeneratedUsingTerminal: EP8309-0022-0021'}
{attribute addProperty BoxType "EP8309-0022-0021"}
{attribute addProperty Id "StatusAT %I*Status_6CCA259F6Rotational_SpeedAT %I*INT2Rotation_DirectionAT %I*UINT2"}
{attribute addProperty CRC "3274820158"}
{attribute addProperty Size "10"}
TYPE TACHO_Single_Shaft_Mode_Input_Channel_C331CA3E EXTENDS InputBase_8311D824 :
STRUCT
	{attribute addProperty Name "Status"}
	Status AT %I* : Status_6CCA259F;
	{attribute addProperty Name "Rotational_Speed"}
	Rotational_Speed AT %I* : INT;
	{attribute addProperty Name "Rotation_Direction"}
	Rotation_Direction AT %I* : UINT;
END_STRUCT
END_TYPE

// ---- DUTs/IO/PDOs/DIG_Inputs_495F5DA4.TcDUT
{attribute 'GeneratedUsingTerminal: EP8309-0022-0021'}
{attribute addProperty BoxType "EP8309-0022-0021"}
{attribute addProperty Id "Digital_Input_X4_Pin4AT %I*BOOL1Digital_Input_X4_Pin2AT %I*BOOL1Digital_Input_X5_Pin4AT %I*BOOL1Digital_Input_X5_Pin2AT %I*BOOL1Digital_Input_X6_Pin4AT %I*BOOL1Digital_Input_X6_Pin2AT %I*BOOL1Digital_Input_X7_Pin4AT %I*BOOL1Digital_Input_X7_Pin2AT %I*BOOL1"}
{attribute addProperty CRC "1230986660"}
{attribute addProperty Size "8"}
TYPE DIG_Inputs_495F5DA4 EXTENDS InputBase_8311D824 :
STRUCT
	{attribute addProperty Name "Digital_Input_X4_Pin4"}
	Digital_Input_X4_Pin4 AT %I* : BOOL;
	{attribute addProperty Name "Digital_Input_X4_Pin2"}
	Digital_Input_X4_Pin2 AT %I* : BOOL;
	{attribute addProperty Name "Digital_Input_X5_Pin4"}
	Digital_Input_X5_Pin4 AT %I* : BOOL;
	{attribute addProperty Name "Digital_Input_X5_Pin2"}
	Digital_Input_X5_Pin2 AT %I* : BOOL;
	{attribute addProperty Name "Digital_Input_X6_Pin4"}
	Digital_Input_X6_Pin4 AT %I* : BOOL;
	{attribute addProperty Name "Digital_Input_X6_Pin2"}
	Digital_Input_X6_Pin2 AT %I* : BOOL;
	{attribute addProperty Name "Digital_Input_X7_Pin4"}
	Digital_Input_X7_Pin4 AT %I* : BOOL;
	{attribute addProperty Name "Digital_Input_X7_Pin2"}
	Digital_Input_X7_Pin2 AT %I* : BOOL;
END_STRUCT
END_TYPE

// ---- DUTs/IO/PDOs/PWM_Status_77939B11.TcDUT
{attribute 'GeneratedUsingTerminal: EP8309-0022-0021'}
{attribute addProperty BoxType "EP8309-0022-0021"}
{attribute addProperty Id "StatusAT %I*Status_72C27E804"}
{attribute addProperty CRC "2006162193"}
{attribute addProperty Size "4"}
TYPE PWM_Status_77939B11 EXTENDS InputBase_8311D824 :
STRUCT
	{attribute addProperty Name "Status"}
	Status AT %I* : Status_72C27E80;
END_STRUCT
END_TYPE

// ---- DUTs/IO/PDOs/DEV_Inputs_FBF180A4.TcDUT
{attribute 'GeneratedUsingTerminal: EP8309-0022-0021'}
{attribute addProperty BoxType "EP8309-0022-0021"}
{attribute addProperty Id "Undervoltage_UsAT %I*BOOL1Undervoltage_UpAT %I*BOOL1"}
{attribute addProperty CRC "4226908324"}
{attribute addProperty Size "2"}
TYPE DEV_Inputs_FBF180A4 EXTENDS InputBase_8311D824 :
STRUCT
	{attribute addProperty Name "Undervoltage_Us"}
	Undervoltage_Us AT %I* : BOOL;
	{attribute addProperty Name "Undervoltage_Up"}
	Undervoltage_Up AT %I* : BOOL;
END_STRUCT
END_TYPE

// ---- DUTs/IO/PDOs/TACHO_Output_Channel_600697D9.TcDUT
{attribute 'GeneratedUsingTerminal: EP8309-0022-0021'}
{attribute addProperty BoxType "EP8309-0022-0021"}
{attribute addProperty Id "Reset_ErrorAT %Q*BOOL1"}
{attribute addProperty CRC "1611044825"}
{attribute addProperty Size "1"}
TYPE TACHO_Output_Channel_600697D9 EXTENDS OutputBase_10CEE7DE :
STRUCT
	{attribute addProperty Name "Reset_Error"}
	Reset_Error AT %Q* : BOOL;
END_STRUCT
END_TYPE

// ---- DUTs/IO/PDOs/DIG_Outputs_0E284394.TcDUT
{attribute 'GeneratedUsingTerminal: EP8309-0022-0021'}
{attribute addProperty BoxType "EP8309-0022-0021"}
{attribute addProperty Id "Digital_Output_X4_Pin4AT %Q*BOOL1Digital_Output_X4_Pin2AT %Q*BOOL1Digital_Output_X5_Pin4AT %Q*BOOL1Digital_Output_X5_Pin2AT %Q*BOOL1Digital_Output_X6_Pin4AT %Q*BOOL1Digital_Output_X6_Pin2AT %Q*BOOL1Digital_Output_X7_Pin4AT %Q*BOOL1Digital_Output_X7_Pin2AT %Q*BOOL1"}
{attribute addProperty CRC "237519764"}
{attribute addProperty Size "8"}
TYPE DIG_Outputs_0E284394 EXTENDS OutputBase_10CEE7DE :
STRUCT
	{attribute addProperty Name "Digital_Output_X4_Pin4"}
	Digital_Output_X4_Pin4 AT %Q* : BOOL;
	{attribute addProperty Name "Digital_Output_X4_Pin2"}
	Digital_Output_X4_Pin2 AT %Q* : BOOL;
	{attribute addProperty Name "Digital_Output_X5_Pin4"}
	Digital_Output_X5_Pin4 AT %Q* : BOOL;
	{attribute addProperty Name "Digital_Output_X5_Pin2"}
	Digital_Output_X5_Pin2 AT %Q* : BOOL;
	{attribute addProperty Name "Digital_Output_X6_Pin4"}
	Digital_Output_X6_Pin4 AT %Q* : BOOL;
	{attribute addProperty Name "Digital_Output_X6_Pin2"}
	Digital_Output_X6_Pin2 AT %Q* : BOOL;
	{attribute addProperty Name "Digital_Output_X7_Pin4"}
	Digital_Output_X7_Pin4 AT %Q* : BOOL;
	{attribute addProperty Name "Digital_Output_X7_Pin2"}
	Digital_Output_X7_Pin2 AT %Q* : BOOL;
END_STRUCT
END_TYPE

// ---- DUTs/IO/PDOs/PWM_Control_63F162E4.TcDUT
{attribute 'GeneratedUsingTerminal: EP8309-0022-0021'}
{attribute addProperty BoxType "EP8309-0022-0021"}
{attribute addProperty Id "ControlAT %Q*Control_254441A53PWM_outputAT %Q*INT2"}
{attribute addProperty CRC "1676763876"}
{attribute addProperty Size "5"}
TYPE PWM_Control_63F162E4 EXTENDS OutputBase_10CEE7DE :
STRUCT
	{attribute addProperty Name "Control"}
	Control AT %Q* : Control_254441A5;
	{attribute addProperty Name "PWM_output"}
	PWM_output AT %Q* : INT;
END_STRUCT
END_TYPE

// ---- DUTs/IO/PDOs/DPO_Inputs_Channel_BF408C57.TcDUT
{attribute 'GeneratedUsingTerminal: EP9214-0023-0019'}
{attribute addProperty BoxType "EP9214-0023-0019"}
{attribute addProperty Id "Error_UsAT %I*BOOL1Error_UpAT %I*BOOL1Warning_UsAT %I*BOOL1Warning_UpAT %I*BOOL1Status_UsAT %I*BOOL1Status_UpAT %I*BOOL1Channel_ErrorAT %I*BOOL1Sync_errorAT %I*BOOL1TxPDO_StateAT %I*BOOL1TxPDO_ToggleAT %I*BOOL1"}
{attribute addProperty CRC "3208678487"}
{attribute addProperty Size "10"}
TYPE DPO_Inputs_Channel_BF408C57 EXTENDS InputBase_8311D824 :
STRUCT
	{attribute addProperty Name "Error_Us"}
	Error_Us AT %I* : BOOL;
	{attribute addProperty Name "Error_Up"}
	Error_Up AT %I* : BOOL;
	{attribute addProperty Name "Warning_Us"}
	Warning_Us AT %I* : BOOL;
	{attribute addProperty Name "Warning_Up"}
	Warning_Up AT %I* : BOOL;
	{attribute addProperty Name "Status_Us"}
	Status_Us AT %I* : BOOL;
	{attribute addProperty Name "Status_Up"}
	Status_Up AT %I* : BOOL;
	{attribute addProperty Name "Channel_Error"}
	Channel_Error AT %I* : BOOL;
	{attribute addProperty Name "Sync_error"}
	Sync_error AT %I* : BOOL;
	{attribute addProperty Name "TxPDO_State"}
	TxPDO_State AT %I* : BOOL;
	{attribute addProperty Name "TxPDO_Toggle"}
	TxPDO_Toggle AT %I* : BOOL;
END_STRUCT
END_TYPE

// ---- DUTs/IO/PDOs/DPO_Inputs_Device_9B08D915.TcDUT
{attribute 'GeneratedUsingTerminal: EP9214-0023-0019'}
{attribute addProperty BoxType "EP9214-0023-0019"}
{attribute addProperty Id "Temperature_WarningAT %I*BOOL1Temperature_ErrorAT %I*BOOL1Us_WarningAT %I*BOOL1Us_ErrorAT %I*BOOL1Up_WarningAT %I*BOOL1Up_ErrorAT %I*BOOL1Global_Error_BitAT %I*BOOL1Reset_InputAT %I*BOOL1TxPDO_StateAT %I*BOOL1TxPDO_ToggleAT %I*BOOL1"}
{attribute addProperty CRC "2601048341"}
{attribute addProperty Size "10"}
TYPE DPO_Inputs_Device_9B08D915 EXTENDS InputBase_8311D824 :
STRUCT
	{attribute addProperty Name "Temperature_Warning"}
	Temperature_Warning AT %I* : BOOL;
	{attribute addProperty Name "Temperature_Error"}
	Temperature_Error AT %I* : BOOL;
	{attribute addProperty Name "Us_Warning"}
	Us_Warning AT %I* : BOOL;
	{attribute addProperty Name "Us_Error"}
	Us_Error AT %I* : BOOL;
	{attribute addProperty Name "Up_Warning"}
	Up_Warning AT %I* : BOOL;
	{attribute addProperty Name "Up_Error"}
	Up_Error AT %I* : BOOL;
	{attribute addProperty Name "Global_Error_Bit"}
	Global_Error_Bit AT %I* : BOOL;
	{attribute addProperty Name "Reset_Input"}
	Reset_Input AT %I* : BOOL;
	{attribute addProperty Name "TxPDO_State"}
	TxPDO_State AT %I* : BOOL;
	{attribute addProperty Name "TxPDO_Toggle"}
	TxPDO_Toggle AT %I* : BOOL;
END_STRUCT
END_TYPE

// ---- DUTs/IO/PDOs/DPO_Outputs_Channel_A459B36C.TcDUT
{attribute 'GeneratedUsingTerminal: EP9214-0023-0019'}
{attribute addProperty BoxType "EP9214-0023-0019"}
{attribute addProperty Id "Output_UsAT %Q*BOOL1Output_UpAT %Q*BOOL1Reset_UsAT %Q*BOOL1Reset_UpAT %Q*BOOL1"}
{attribute addProperty CRC "2757342060"}
{attribute addProperty Size "4"}
TYPE DPO_Outputs_Channel_A459B36C EXTENDS OutputBase_10CEE7DE :
STRUCT
	{attribute addProperty Name "Output_Us"}
	Output_Us AT %Q* : BOOL;
	{attribute addProperty Name "Output_Up"}
	Output_Up AT %Q* : BOOL;
	{attribute addProperty Name "Reset_Us"}
	Reset_Us AT %Q* : BOOL;
	{attribute addProperty Name "Reset_Up"}
	Reset_Up AT %Q* : BOOL;
END_STRUCT
END_TYPE

// ---- DUTs/IO/PDOs/DPO_Outputs_Device_B673A337.TcDUT
{attribute 'GeneratedUsingTerminal: EP9214-0023-0019'}
{attribute addProperty BoxType "EP9214-0023-0019"}
{attribute addProperty Id "Enable_Control_Via_FieldbusAT %Q*BOOL1Global_ResetAT %Q*BOOL1"}
{attribute addProperty CRC "3061031735"}
{attribute addProperty Size "2"}
TYPE DPO_Outputs_Device_B673A337 EXTENDS OutputBase_10CEE7DE :
STRUCT
	{attribute addProperty Name "Enable_Control_Via_Fieldbus"}
	Enable_Control_Via_Fieldbus AT %Q* : BOOL;
	{attribute addProperty Name "Global_Reset"}
	Global_Reset AT %Q* : BOOL;
END_STRUCT
END_TYPE

// ---- DUTs/IO/PDOs/DPO_Inputs_Channel_F87663B8.TcDUT
{attribute 'GeneratedUsingTerminal: EP9224-0023-0016'}
{attribute addProperty BoxType "EP9224-0023-0016"}
{attribute addProperty Id "Error_UsAT %I*BOOL1Error_UpAT %I*BOOL1Warning_UsAT %I*BOOL1Warning_UpAT %I*BOOL1Status_UsAT %I*BOOL1Status_UpAT %I*BOOL1Channel_ErrorAT %I*BOOL1Error_Sum_CurrentAT %I*BOOL1Warning_Sum_CurrentAT %I*BOOL1TxPDO_StateAT %I*BOOL1TxPDO_ToggleAT %I*BOOL1Current_UsAT %I*INT2Current_UpAT %I*INT2"}
{attribute addProperty CRC "4168508344"}
{attribute addProperty Size "15"}
TYPE DPO_Inputs_Channel_F87663B8 EXTENDS InputBase_8311D824 :
STRUCT
	{attribute addProperty Name "Error_Us"}
	Error_Us AT %I* : BOOL;
	{attribute addProperty Name "Error_Up"}
	Error_Up AT %I* : BOOL;
	{attribute addProperty Name "Warning_Us"}
	Warning_Us AT %I* : BOOL;
	{attribute addProperty Name "Warning_Up"}
	Warning_Up AT %I* : BOOL;
	{attribute addProperty Name "Status_Us"}
	Status_Us AT %I* : BOOL;
	{attribute addProperty Name "Status_Up"}
	Status_Up AT %I* : BOOL;
	{attribute addProperty Name "Channel_Error"}
	Channel_Error AT %I* : BOOL;
	{attribute addProperty Name "Error_Sum_Current"}
	Error_Sum_Current AT %I* : BOOL;
	{attribute addProperty Name "Warning_Sum_Current"}
	Warning_Sum_Current AT %I* : BOOL;
	{attribute addProperty Name "TxPDO_State"}
	TxPDO_State AT %I* : BOOL;
	{attribute addProperty Name "TxPDO_Toggle"}
	TxPDO_Toggle AT %I* : BOOL;
	{attribute addProperty Name "Current_Us"}
	Current_Us AT %I* : INT;
	{attribute addProperty Name "Current_Up"}
	Current_Up AT %I* : INT;
END_STRUCT
END_TYPE

// ---- DUTs/IO/PDOs/DPO_Inputs_Device_99241EEA.TcDUT
{attribute 'GeneratedUsingTerminal: EP9224-0023-0016'}
{attribute addProperty BoxType "EP9224-0023-0016"}
{attribute addProperty Id "Temperature_WarningAT %I*BOOL1Temperature_ErrorAT %I*BOOL1Us_WarningAT %I*BOOL1Us_ErrorAT %I*BOOL1Up_WarningAT %I*BOOL1Up_ErrorAT %I*BOOL1Global_Error_BitAT %I*BOOL1Sum_Current_WarningAT %I*BOOL1Sum_Current_ErrorAT %I*BOOL1Reset_InputAT %I*BOOL1TxPDO_StateAT %I*BOOL1TxPDO_ToggleAT %I*BOOL1Current_UsAT %I*INT2Current_UpAT %I*INT2Voltage_UsAT %I*INT2Voltage_UpAT %I*INT2TemperatureAT %I*INT2"}
{attribute addProperty CRC "2569281258"}
{attribute addProperty Size "22"}
TYPE DPO_Inputs_Device_99241EEA EXTENDS InputBase_8311D824 :
STRUCT
	{attribute addProperty Name "Temperature_Warning"}
	Temperature_Warning AT %I* : BOOL;
	{attribute addProperty Name "Temperature_Error"}
	Temperature_Error AT %I* : BOOL;
	{attribute addProperty Name "Us_Warning"}
	Us_Warning AT %I* : BOOL;
	{attribute addProperty Name "Us_Error"}
	Us_Error AT %I* : BOOL;
	{attribute addProperty Name "Up_Warning"}
	Up_Warning AT %I* : BOOL;
	{attribute addProperty Name "Up_Error"}
	Up_Error AT %I* : BOOL;
	{attribute addProperty Name "Global_Error_Bit"}
	Global_Error_Bit AT %I* : BOOL;
	{attribute addProperty Name "Sum_Current_Warning"}
	Sum_Current_Warning AT %I* : BOOL;
	{attribute addProperty Name "Sum_Current_Error"}
	Sum_Current_Error AT %I* : BOOL;
	{attribute addProperty Name "Reset_Input"}
	Reset_Input AT %I* : BOOL;
	{attribute addProperty Name "TxPDO_State"}
	TxPDO_State AT %I* : BOOL;
	{attribute addProperty Name "TxPDO_Toggle"}
	TxPDO_Toggle AT %I* : BOOL;
	{attribute addProperty Name "Current_Us"}
	Current_Us AT %I* : INT;
	{attribute addProperty Name "Current_Up"}
	Current_Up AT %I* : INT;
	{attribute addProperty Name "Voltage_Us"}
	Voltage_Us AT %I* : INT;
	{attribute addProperty Name "Voltage_Up"}
	Voltage_Up AT %I* : INT;
	{attribute addProperty Name "Temperature"}
	Temperature AT %I* : INT;
END_STRUCT
END_TYPE

// ---- DUTs/IO/PDOs/BCT_Inputs_7ACE8FA6.TcDUT
{attribute 'GeneratedUsingTerminal: EP9576-1032-0016'}
{attribute addProperty BoxType "EP9576-1032-0016"}
{attribute addProperty Id "Terminal_OvertemperatureAT %I*BOOL1I2T_errorAT %I*BOOL1I2T_warningAT %I*BOOL1OvervoltageAT %I*BOOL1UndervoltageAT %I*BOOL1Chopper_onAT %I*BOOL1Overcurrent_ProtectionAT %I*BOOL1Input_cycle_counterAT %I*BYTE1DC_link_voltageAT %I*UDINT4Resistor_CurrentAT %I*DINT4Duty_CycleAT %I*USINT1"}
{attribute addProperty CRC "2060357542"}
{attribute addProperty Size "17"}
TYPE BCT_Inputs_7ACE8FA6 EXTENDS InputBase_8311D824 :
STRUCT
	{attribute addProperty Name "Terminal_Overtemperature"}
	Terminal_Overtemperature AT %I* : BOOL;
	{attribute addProperty Name "I2T_error"}
	I2T_error AT %I* : BOOL;
	{attribute addProperty Name "I2T_warning"}
	I2T_warning AT %I* : BOOL;
	{attribute addProperty Name "Overvoltage"}
	Overvoltage AT %I* : BOOL;
	{attribute addProperty Name "Undervoltage"}
	Undervoltage AT %I* : BOOL;
	{attribute addProperty Name "Chopper_on"}
	Chopper_on AT %I* : BOOL;
	{attribute addProperty Name "Overcurrent_Protection"}
	Overcurrent_Protection AT %I* : BOOL;
	{attribute addProperty Name "Input_cycle_counter"}
	Input_cycle_counter AT %I* : BYTE;
	{attribute addProperty Name "DC_link_voltage"}
	DC_link_voltage AT %I* : UDINT;
	{attribute addProperty Name "Resistor_Current"}
	Resistor_Current AT %I* : DINT;
	{attribute addProperty Name "Duty_Cycle"}
	Duty_Cycle AT %I* : USINT;
END_STRUCT
END_TYPE

// ---- DUTs/IO/PDOs/DPO_Inputs_Channel_0E6D6BE5.TcDUT
{attribute 'GeneratedUsingTerminal: EP9224-0037-0017'}
{attribute addProperty BoxType "EP9224-0037-0017"}
{attribute addProperty Id "StatusAT %I*Status_15ACD20111Current_UsAT %I*INT2Current_UpAT %I*INT2"}
{attribute addProperty CRC "242052069"}
{attribute addProperty Size "15"}
TYPE DPO_Inputs_Channel_0E6D6BE5 EXTENDS InputBase_8311D824 :
STRUCT
	{attribute addProperty Name "Status"}
	Status AT %I* : Status_15ACD201;
	{attribute addProperty Name "Current_Us"}
	Current_Us AT %I* : INT;
	{attribute addProperty Name "Current_Up"}
	Current_Up AT %I* : INT;
END_STRUCT
END_TYPE

// ---- DUTs/IO/PDOs/DPO_Inputs_Device_0C16AFA0.TcDUT
{attribute 'GeneratedUsingTerminal: EP9224-0037-0017'}
{attribute addProperty BoxType "EP9224-0037-0017"}
{attribute addProperty Id "Device_StatusAT %I*Device_Status_033C68E911Current_UsAT %I*INT2Current_UpAT %I*INT2Voltage_UsAT %I*INT2Voltage_UpAT %I*INT2TemperatureAT %I*INT2"}
{attribute addProperty CRC "202813344"}
{attribute addProperty Size "21"}
TYPE DPO_Inputs_Device_0C16AFA0 EXTENDS InputBase_8311D824 :
STRUCT
	{attribute addProperty Name "Device_Status"}
	Device_Status AT %I* : Device_Status_033C68E9;
	{attribute addProperty Name "Current_Us"}
	Current_Us AT %I* : INT;
	{attribute addProperty Name "Current_Up"}
	Current_Up AT %I* : INT;
	{attribute addProperty Name "Voltage_Us"}
	Voltage_Us AT %I* : INT;
	{attribute addProperty Name "Voltage_Up"}
	Voltage_Up AT %I* : INT;
	{attribute addProperty Name "Temperature"}
	Temperature AT %I* : INT;
END_STRUCT
END_TYPE

// ---- DUTs/IO/PDOs/InfoData_E68C61CD.TcDUT
{attribute 'GeneratedUsingTerminal: IODEVICETYPE_ETHERCATPROT'}
{attribute addProperty BoxType "IODEVICETYPE_ETHERCATPROT"}
{attribute addProperty Id "ChangeCountAT %I*UINT2DevIdAT %I*UINT2AmsNetIdAT %I*AMSNETID6CfgSlaveCountAT %I*UINT2DcToTcTimeOffsetAT %I*LINT8DcToExtTimeOffsetAT %I*LINT8"}
{attribute addProperty CRC "3867959757"}
{attribute addProperty Size "28"}
TYPE InfoData_E68C61CD EXTENDS InputBase_8311D824 :
STRUCT
	{attribute addProperty Name "ChangeCount"}
	ChangeCount AT %I* : UINT;
	{attribute addProperty Name "DevId"}
	DevId AT %I* : UINT;
	{attribute addProperty Name "AmsNetId"}
	AmsNetId AT %I* : AMSNETID;
	{attribute addProperty Name "CfgSlaveCount"}
	CfgSlaveCount AT %I* : UINT;
	{attribute addProperty Name "DcToTcTimeOffset"}
	DcToTcTimeOffset AT %I* : LINT;
	{attribute addProperty Name "DcToExtTimeOffset"}
	DcToExtTimeOffset AT %I* : LINT;
END_STRUCT
END_TYPE

// ---- DUTs/IO/PDOs/InfoData_2A97D6CF.TcDUT
{attribute 'GeneratedUsingTerminal: IODEVICETYPE_ETHERCATPROT'}
{attribute addProperty BoxType "IODEVICETYPE_ETHERCATPROT"}
{attribute addProperty Id "ObjectIdAT %I*OTCID4StateAT %I*UINT2SlaveCountAT %I*UINT2"}
{attribute addProperty CRC "714593999"}
{attribute addProperty Size "8"}
TYPE InfoData_2A97D6CF EXTENDS InputBase_8311D824 :
STRUCT
	{attribute addProperty Name "ObjectId"}
	ObjectId AT %I* : OTCID;
	{attribute addProperty Name "State"}
	State AT %I* : UINT;
	{attribute addProperty Name "SlaveCount"}
	SlaveCount AT %I* : UINT;
END_STRUCT
END_TYPE

// ---- DUTs/IO/PDOs/Inputs_25A0042B.TcDUT
{attribute 'GeneratedUsingTerminal: IODEVICETYPE_ETHERCATPROT'}
{attribute addProperty BoxType "IODEVICETYPE_ETHERCATPROT"}
{attribute addProperty Id "SlaveCountAT %I*UINT2DevStateAT %I*UINT2Frm0StateAT %I*UINT2Frm0WcStateAT %I*UINT2Frm0InputToggleAT %I*UINT2Frm1StateAT %I*UINT2Frm1WcStateAT %I*UINT2Frm1InputToggleAT %I*UINT2Frm2StateAT %I*UINT2Frm2WcStateAT %I*UINT2Frm2InputToggleAT %I*UINT2Frm3StateAT %I*UINT2Frm3WcStateAT %I*UINT2Frm3InputToggleAT %I*UINT2Frm4StateAT %I*UINT2Frm4WcStateAT %I*UINT2Frm4InputToggleAT %I*UINT2Frm5StateAT %I*UINT2Frm5WcStateAT %I*UINT2Frm5InputToggleAT %I*UINT2Frm6StateAT %I*UINT2Frm6WcStateAT %I*UINT2Frm6InputToggleAT %I*UINT2Frm7StateAT %I*UINT2Frm7WcStateAT %I*UINT2Frm7InputToggleAT %I*UINT2Frm8StateAT %I*UINT2Frm8WcStateAT %I*UINT2Frm8InputToggleAT %I*UINT2Frm9StateAT %I*UINT2Frm9WcStateAT %I*UINT2Frm9InputToggleAT %I*UINT2Frm10StateAT %I*UINT2Frm10WcStateAT %I*UINT2Frm10InputToggleAT %I*UINT2Frm11StateAT %I*UINT2Frm11WcStateAT %I*UINT2Frm11InputToggleAT %I*UINT2Frm12StateAT %I*UINT2Frm12WcStateAT %I*UINT2Frm12InputToggleAT %I*UINT2Frm13StateAT %I*UINT2Frm13WcStateAT %I*UINT2Frm13InputToggleAT %I*UINT2Frm14StateAT %I*UINT2Frm14WcStateAT %I*UINT2Frm14InputToggleAT %I*UINT2Frm15StateAT %I*UINT2Frm15WcStateAT %I*UINT2Frm15InputToggleAT %I*UINT2Frm16StateAT %I*UINT2Frm16WcStateAT %I*UINT2Frm16InputToggleAT %I*UINT2Frm17StateAT %I*UINT2Frm17WcStateAT %I*UINT2Frm17InputToggleAT %I*UINT2Frm18StateAT %I*UINT2Frm18WcStateAT %I*UINT2Frm18InputToggleAT %I*UINT2Frm19StateAT %I*UINT2Frm19WcStateAT %I*UINT2Frm19InputToggleAT %I*UINT2Frm20StateAT %I*UINT2Frm20WcStateAT %I*UINT2Frm20InputToggleAT %I*UINT2Frm21StateAT %I*UINT2Frm21WcStateAT %I*UINT2Frm21InputToggleAT %I*UINT2Frm22StateAT %I*UINT2Frm22WcStateAT %I*UINT2Frm22InputToggleAT %I*UINT2Frm23StateAT %I*UINT2Frm23WcStateAT %I*UINT2Frm23InputToggleAT %I*UINT2Frm24StateAT %I*UINT2Frm24WcStateAT %I*UINT2Frm24InputToggleAT %I*UINT2Frm25StateAT %I*UINT2Frm25WcStateAT %I*UINT2Frm25InputToggleAT %I*UINT2"}
{attribute addProperty CRC "631243819"}
{attribute addProperty Size "160"}
TYPE Inputs_25A0042B EXTENDS InputBase_8311D824 :
STRUCT
	{attribute addProperty Name "SlaveCount"}
	SlaveCount AT %I* : UINT;
	{attribute addProperty Name "DevState"}
	DevState AT %I* : UINT;
	{attribute addProperty Name "Frm0State"}
	Frm0State AT %I* : UINT;
	{attribute addProperty Name "Frm0WcState"}
	Frm0WcState AT %I* : UINT;
	{attribute addProperty Name "Frm0InputToggle"}
	Frm0InputToggle AT %I* : UINT;
	{attribute addProperty Name "Frm1State"}
	Frm1State AT %I* : UINT;
	{attribute addProperty Name "Frm1WcState"}
	Frm1WcState AT %I* : UINT;
	{attribute addProperty Name "Frm1InputToggle"}
	Frm1InputToggle AT %I* : UINT;
	{attribute addProperty Name "Frm2State"}
	Frm2State AT %I* : UINT;
	{attribute addProperty Name "Frm2WcState"}
	Frm2WcState AT %I* : UINT;
	{attribute addProperty Name "Frm2InputToggle"}
	Frm2InputToggle AT %I* : UINT;
	{attribute addProperty Name "Frm3State"}
	Frm3State AT %I* : UINT;
	{attribute addProperty Name "Frm3WcState"}
	Frm3WcState AT %I* : UINT;
	{attribute addProperty Name "Frm3InputToggle"}
	Frm3InputToggle AT %I* : UINT;
	{attribute addProperty Name "Frm4State"}
	Frm4State AT %I* : UINT;
	{attribute addProperty Name "Frm4WcState"}
	Frm4WcState AT %I* : UINT;
	{attribute addProperty Name "Frm4InputToggle"}
	Frm4InputToggle AT %I* : UINT;
	{attribute addProperty Name "Frm5State"}
	Frm5State AT %I* : UINT;
	{attribute addProperty Name "Frm5WcState"}
	Frm5WcState AT %I* : UINT;
	{attribute addProperty Name "Frm5InputToggle"}
	Frm5InputToggle AT %I* : UINT;
	{attribute addProperty Name "Frm6State"}
	Frm6State AT %I* : UINT;
	{attribute addProperty Name "Frm6WcState"}
	Frm6WcState AT %I* : UINT;
	{attribute addProperty Name "Frm6InputToggle"}
	Frm6InputToggle AT %I* : UINT;
	{attribute addProperty Name "Frm7State"}
	Frm7State AT %I* : UINT;
	{attribute addProperty Name "Frm7WcState"}
	Frm7WcState AT %I* : UINT;
	{attribute addProperty Name "Frm7InputToggle"}
	Frm7InputToggle AT %I* : UINT;
	{attribute addProperty Name "Frm8State"}
	Frm8State AT %I* : UINT;
	{attribute addProperty Name "Frm8WcState"}
	Frm8WcState AT %I* : UINT;
	{attribute addProperty Name "Frm8InputToggle"}
	Frm8InputToggle AT %I* : UINT;
	{attribute addProperty Name "Frm9State"}
	Frm9State AT %I* : UINT;
	{attribute addProperty Name "Frm9WcState"}
	Frm9WcState AT %I* : UINT;
	{attribute addProperty Name "Frm9InputToggle"}
	Frm9InputToggle AT %I* : UINT;
	{attribute addProperty Name "Frm10State"}
	Frm10State AT %I* : UINT;
	{attribute addProperty Name "Frm10WcState"}
	Frm10WcState AT %I* : UINT;
	{attribute addProperty Name "Frm10InputToggle"}
	Frm10InputToggle AT %I* : UINT;
	{attribute addProperty Name "Frm11State"}
	Frm11State AT %I* : UINT;
	{attribute addProperty Name "Frm11WcState"}
	Frm11WcState AT %I* : UINT;
	{attribute addProperty Name "Frm11InputToggle"}
	Frm11InputToggle AT %I* : UINT;
	{attribute addProperty Name "Frm12State"}
	Frm12State AT %I* : UINT;
	{attribute addProperty Name "Frm12WcState"}
	Frm12WcState AT %I* : UINT;
	{attribute addProperty Name "Frm12InputToggle"}
	Frm12InputToggle AT %I* : UINT;
	{attribute addProperty Name "Frm13State"}
	Frm13State AT %I* : UINT;
	{attribute addProperty Name "Frm13WcState"}
	Frm13WcState AT %I* : UINT;
	{attribute addProperty Name "Frm13InputToggle"}
	Frm13InputToggle AT %I* : UINT;
	{attribute addProperty Name "Frm14State"}
	Frm14State AT %I* : UINT;
	{attribute addProperty Name "Frm14WcState"}
	Frm14WcState AT %I* : UINT;
	{attribute addProperty Name "Frm14InputToggle"}
	Frm14InputToggle AT %I* : UINT;
	{attribute addProperty Name "Frm15State"}
	Frm15State AT %I* : UINT;
	{attribute addProperty Name "Frm15WcState"}
	Frm15WcState AT %I* : UINT;
	{attribute addProperty Name "Frm15InputToggle"}
	Frm15InputToggle AT %I* : UINT;
	{attribute addProperty Name "Frm16State"}
	Frm16State AT %I* : UINT;
	{attribute addProperty Name "Frm16WcState"}
	Frm16WcState AT %I* : UINT;
	{attribute addProperty Name "Frm16InputToggle"}
	Frm16InputToggle AT %I* : UINT;
	{attribute addProperty Name "Frm17State"}
	Frm17State AT %I* : UINT;
	{attribute addProperty Name "Frm17WcState"}
	Frm17WcState AT %I* : UINT;
	{attribute addProperty Name "Frm17InputToggle"}
	Frm17InputToggle AT %I* : UINT;
	{attribute addProperty Name "Frm18State"}
	Frm18State AT %I* : UINT;
	{attribute addProperty Name "Frm18WcState"}
	Frm18WcState AT %I* : UINT;
	{attribute addProperty Name "Frm18InputToggle"}
	Frm18InputToggle AT %I* : UINT;
	{attribute addProperty Name "Frm19State"}
	Frm19State AT %I* : UINT;
	{attribute addProperty Name "Frm19WcState"}
	Frm19WcState AT %I* : UINT;
	{attribute addProperty Name "Frm19InputToggle"}
	Frm19InputToggle AT %I* : UINT;
	{attribute addProperty Name "Frm20State"}
	Frm20State AT %I* : UINT;
	{attribute addProperty Name "Frm20WcState"}
	Frm20WcState AT %I* : UINT;
	{attribute addProperty Name "Frm20InputToggle"}
	Frm20InputToggle AT %I* : UINT;
	{attribute addProperty Name "Frm21State"}
	Frm21State AT %I* : UINT;
	{attribute addProperty Name "Frm21WcState"}
	Frm21WcState AT %I* : UINT;
	{attribute addProperty Name "Frm21InputToggle"}
	Frm21InputToggle AT %I* : UINT;
	{attribute addProperty Name "Frm22State"}
	Frm22State AT %I* : UINT;
	{attribute addProperty Name "Frm22WcState"}
	Frm22WcState AT %I* : UINT;
	{attribute addProperty Name "Frm22InputToggle"}
	Frm22InputToggle AT %I* : UINT;
	{attribute addProperty Name "Frm23State"}
	Frm23State AT %I* : UINT;
	{attribute addProperty Name "Frm23WcState"}
	Frm23WcState AT %I* : UINT;
	{attribute addProperty Name "Frm23InputToggle"}
	Frm23InputToggle AT %I* : UINT;
	{attribute addProperty Name "Frm24State"}
	Frm24State AT %I* : UINT;
	{attribute addProperty Name "Frm24WcState"}
	Frm24WcState AT %I* : UINT;
	{attribute addProperty Name "Frm24InputToggle"}
	Frm24InputToggle AT %I* : UINT;
	{attribute addProperty Name "Frm25State"}
	Frm25State AT %I* : UINT;
	{attribute addProperty Name "Frm25WcState"}
	Frm25WcState AT %I* : UINT;
	{attribute addProperty Name "Frm25InputToggle"}
	Frm25InputToggle AT %I* : UINT;
END_STRUCT
END_TYPE

// ---- DUTs/IO/PDOs/Outputs_2397A10E.TcDUT
{attribute 'GeneratedUsingTerminal: IODEVICETYPE_ETHERCATPROT'}
{attribute addProperty BoxType "IODEVICETYPE_ETHERCATPROT"}
{attribute addProperty Id "DevCtrlAT %Q*UINT2Frm0CtrlAT %Q*UINT2Frm0WcCtrlAT %Q*UINT2Frm1CtrlAT %Q*UINT2Frm1WcCtrlAT %Q*UINT2Frm2CtrlAT %Q*UINT2Frm2WcCtrlAT %Q*UINT2Frm3CtrlAT %Q*UINT2Frm3WcCtrlAT %Q*UINT2Frm4CtrlAT %Q*UINT2Frm4WcCtrlAT %Q*UINT2Frm5CtrlAT %Q*UINT2Frm5WcCtrlAT %Q*UINT2Frm6CtrlAT %Q*UINT2Frm6WcCtrlAT %Q*UINT2Frm7CtrlAT %Q*UINT2Frm7WcCtrlAT %Q*UINT2Frm8CtrlAT %Q*UINT2Frm8WcCtrlAT %Q*UINT2Frm9CtrlAT %Q*UINT2Frm9WcCtrlAT %Q*UINT2Frm10CtrlAT %Q*UINT2Frm10WcCtrlAT %Q*UINT2Frm11CtrlAT %Q*UINT2Frm11WcCtrlAT %Q*UINT2Frm12CtrlAT %Q*UINT2Frm12WcCtrlAT %Q*UINT2Frm13CtrlAT %Q*UINT2Frm13WcCtrlAT %Q*UINT2Frm14CtrlAT %Q*UINT2Frm14WcCtrlAT %Q*UINT2Frm15CtrlAT %Q*UINT2Frm15WcCtrlAT %Q*UINT2Frm16CtrlAT %Q*UINT2Frm16WcCtrlAT %Q*UINT2Frm17CtrlAT %Q*UINT2Frm17WcCtrlAT %Q*UINT2Frm18CtrlAT %Q*UINT2Frm18WcCtrlAT %Q*UINT2Frm19CtrlAT %Q*UINT2Frm19WcCtrlAT %Q*UINT2Frm20CtrlAT %Q*UINT2Frm20WcCtrlAT %Q*UINT2Frm21CtrlAT %Q*UINT2Frm21WcCtrlAT %Q*UINT2Frm22CtrlAT %Q*UINT2Frm22WcCtrlAT %Q*UINT2Frm23CtrlAT %Q*UINT2Frm23WcCtrlAT %Q*UINT2Frm24CtrlAT %Q*UINT2Frm24WcCtrlAT %Q*UINT2Frm25CtrlAT %Q*UINT2Frm25WcCtrlAT %Q*UINT2"}
{attribute addProperty CRC "597139726"}
{attribute addProperty Size "106"}
TYPE Outputs_2397A10E EXTENDS OutputBase_10CEE7DE :
STRUCT
	{attribute addProperty Name "DevCtrl"}
	DevCtrl AT %Q* : UINT;
	{attribute addProperty Name "Frm0Ctrl"}
	Frm0Ctrl AT %Q* : UINT;
	{attribute addProperty Name "Frm0WcCtrl"}
	Frm0WcCtrl AT %Q* : UINT;
	{attribute addProperty Name "Frm1Ctrl"}
	Frm1Ctrl AT %Q* : UINT;
	{attribute addProperty Name "Frm1WcCtrl"}
	Frm1WcCtrl AT %Q* : UINT;
	{attribute addProperty Name "Frm2Ctrl"}
	Frm2Ctrl AT %Q* : UINT;
	{attribute addProperty Name "Frm2WcCtrl"}
	Frm2WcCtrl AT %Q* : UINT;
	{attribute addProperty Name "Frm3Ctrl"}
	Frm3Ctrl AT %Q* : UINT;
	{attribute addProperty Name "Frm3WcCtrl"}
	Frm3WcCtrl AT %Q* : UINT;
	{attribute addProperty Name "Frm4Ctrl"}
	Frm4Ctrl AT %Q* : UINT;
	{attribute addProperty Name "Frm4WcCtrl"}
	Frm4WcCtrl AT %Q* : UINT;
	{attribute addProperty Name "Frm5Ctrl"}
	Frm5Ctrl AT %Q* : UINT;
	{attribute addProperty Name "Frm5WcCtrl"}
	Frm5WcCtrl AT %Q* : UINT;
	{attribute addProperty Name "Frm6Ctrl"}
	Frm6Ctrl AT %Q* : UINT;
	{attribute addProperty Name "Frm6WcCtrl"}
	Frm6WcCtrl AT %Q* : UINT;
	{attribute addProperty Name "Frm7Ctrl"}
	Frm7Ctrl AT %Q* : UINT;
	{attribute addProperty Name "Frm7WcCtrl"}
	Frm7WcCtrl AT %Q* : UINT;
	{attribute addProperty Name "Frm8Ctrl"}
	Frm8Ctrl AT %Q* : UINT;
	{attribute addProperty Name "Frm8WcCtrl"}
	Frm8WcCtrl AT %Q* : UINT;
	{attribute addProperty Name "Frm9Ctrl"}
	Frm9Ctrl AT %Q* : UINT;
	{attribute addProperty Name "Frm9WcCtrl"}
	Frm9WcCtrl AT %Q* : UINT;
	{attribute addProperty Name "Frm10Ctrl"}
	Frm10Ctrl AT %Q* : UINT;
	{attribute addProperty Name "Frm10WcCtrl"}
	Frm10WcCtrl AT %Q* : UINT;
	{attribute addProperty Name "Frm11Ctrl"}
	Frm11Ctrl AT %Q* : UINT;
	{attribute addProperty Name "Frm11WcCtrl"}
	Frm11WcCtrl AT %Q* : UINT;
	{attribute addProperty Name "Frm12Ctrl"}
	Frm12Ctrl AT %Q* : UINT;
	{attribute addProperty Name "Frm12WcCtrl"}
	Frm12WcCtrl AT %Q* : UINT;
	{attribute addProperty Name "Frm13Ctrl"}
	Frm13Ctrl AT %Q* : UINT;
	{attribute addProperty Name "Frm13WcCtrl"}
	Frm13WcCtrl AT %Q* : UINT;
	{attribute addProperty Name "Frm14Ctrl"}
	Frm14Ctrl AT %Q* : UINT;
	{attribute addProperty Name "Frm14WcCtrl"}
	Frm14WcCtrl AT %Q* : UINT;
	{attribute addProperty Name "Frm15Ctrl"}
	Frm15Ctrl AT %Q* : UINT;
	{attribute addProperty Name "Frm15WcCtrl"}
	Frm15WcCtrl AT %Q* : UINT;
	{attribute addProperty Name "Frm16Ctrl"}
	Frm16Ctrl AT %Q* : UINT;
	{attribute addProperty Name "Frm16WcCtrl"}
	Frm16WcCtrl AT %Q* : UINT;
	{attribute addProperty Name "Frm17Ctrl"}
	Frm17Ctrl AT %Q* : UINT;
	{attribute addProperty Name "Frm17WcCtrl"}
	Frm17WcCtrl AT %Q* : UINT;
	{attribute addProperty Name "Frm18Ctrl"}
	Frm18Ctrl AT %Q* : UINT;
	{attribute addProperty Name "Frm18WcCtrl"}
	Frm18WcCtrl AT %Q* : UINT;
	{attribute addProperty Name "Frm19Ctrl"}
	Frm19Ctrl AT %Q* : UINT;
	{attribute addProperty Name "Frm19WcCtrl"}
	Frm19WcCtrl AT %Q* : UINT;
	{attribute addProperty Name "Frm20Ctrl"}
	Frm20Ctrl AT %Q* : UINT;
	{attribute addProperty Name "Frm20WcCtrl"}
	Frm20WcCtrl AT %Q* : UINT;
	{attribute addProperty Name "Frm21Ctrl"}
	Frm21Ctrl AT %Q* : UINT;
	{attribute addProperty Name "Frm21WcCtrl"}
	Frm21WcCtrl AT %Q* : UINT;
	{attribute addProperty Name "Frm22Ctrl"}
	Frm22Ctrl AT %Q* : UINT;
	{attribute addProperty Name "Frm22WcCtrl"}
	Frm22WcCtrl AT %Q* : UINT;
	{attribute addProperty Name "Frm23Ctrl"}
	Frm23Ctrl AT %Q* : UINT;
	{attribute addProperty Name "Frm23WcCtrl"}
	Frm23WcCtrl AT %Q* : UINT;
	{attribute addProperty Name "Frm24Ctrl"}
	Frm24Ctrl AT %Q* : UINT;
	{attribute addProperty Name "Frm24WcCtrl"}
	Frm24WcCtrl AT %Q* : UINT;
	{attribute addProperty Name "Frm25Ctrl"}
	Frm25Ctrl AT %Q* : UINT;
	{attribute addProperty Name "Frm25WcCtrl"}
	Frm25WcCtrl AT %Q* : UINT;
END_STRUCT
END_TYPE

// ---- DUTs/IO/Boxes/EK1100_1FC0878B.TcDUT
{attribute 'GeneratedUsingTerminal: EK1100-0000-0018'}
{attribute addProperty BoxType "EK1100-0000-0018"}
{attribute addProperty Description "EK1100 EtherCAT Coupler (2A E-Bus)"}
{attribute addProperty Physics "YKY"}
{attribute addProperty Id "InfoDataAT %I*InfoData_6F19DB2B2"}
{attribute addProperty CRC "532711307"}
{attribute addProperty Size "2"}
TYPE EK1100_1FC0878B EXTENDS EtcSlaveBoxBase_77A0E4A7 :
STRUCT
	{attribute addProperty Name "InfoData"}
	InfoData : InfoData_6F19DB2B;
END_STRUCT
END_TYPE

// ---- DUTs/IO/Boxes/EK1122_1FC0878B.TcDUT
{attribute 'GeneratedUsingTerminal: EK1122-0000-0018'}
{attribute addProperty BoxType "EK1122-0000-0018"}
{attribute addProperty Description "EK1122 2 port EtherCAT junction"}
{attribute addProperty Physics "KYKY"}
{attribute addProperty Id "InfoDataAT %I*InfoData_6F19DB2B2"}
{attribute addProperty CRC "532711307"}
{attribute addProperty Size "2"}
TYPE EK1122_1FC0878B EXTENDS EtcSlaveTerminalBase_947E5A46 :
STRUCT
	{attribute addProperty Name "InfoData"}
	InfoData : InfoData_6F19DB2B;
END_STRUCT
END_TYPE

// ---- DUTs/IO/Boxes/EP1008_78E8D3DD.TcDUT
{attribute 'GeneratedUsingTerminal: EP1008-0001-0016'}
{attribute addProperty BoxType "EP1008-0001-0016"}
{attribute addProperty Description "EP1008-0001 8 Ch. Dig. Input 24V, 3ms, M8"}
{attribute addProperty Physics "YY"}
{attribute addProperty Id "Channel_1AT %I*Channel_830843C11Channel_2AT %I*Channel_830843C11Channel_3AT %I*Channel_830843C11Channel_4AT %I*Channel_830843C11Channel_5AT %I*Channel_830843C11Channel_6AT %I*Channel_830843C11Channel_7AT %I*Channel_830843C11Channel_8AT %I*Channel_830843C11WcStateAT %I*WcState_9091E0EB2InfoDataAT %I*InfoData_6F19DB2B2"}
{attribute addProperty CRC "2028524509"}
{attribute addProperty Size "12"}
TYPE EP1008_78E8D3DD EXTENDS EtcSlaveBoxBase_77A0E4A7 :
STRUCT
	{attribute addProperty Name "Channel_1"}
	Channel_1 : Channel_830843C1;
	{attribute addProperty Name "Channel_2"}
	Channel_2 : Channel_830843C1;
	{attribute addProperty Name "Channel_3"}
	Channel_3 : Channel_830843C1;
	{attribute addProperty Name "Channel_4"}
	Channel_4 : Channel_830843C1;
	{attribute addProperty Name "Channel_5"}
	Channel_5 : Channel_830843C1;
	{attribute addProperty Name "Channel_6"}
	Channel_6 : Channel_830843C1;
	{attribute addProperty Name "Channel_7"}
	Channel_7 : Channel_830843C1;
	{attribute addProperty Name "Channel_8"}
	Channel_8 : Channel_830843C1;
	{attribute addProperty Name "WcState"}
	WcState : WcState_9091E0EB;
	{attribute addProperty Name "InfoData"}
	InfoData : InfoData_6F19DB2B;
END_STRUCT
END_TYPE

// ---- DUTs/IO/Boxes/EP1018_78E8D3DD.TcDUT
{attribute 'GeneratedUsingTerminal: EP1018-0001-0016'}
{attribute addProperty BoxType "EP1018-0001-0016"}
{attribute addProperty Description "EP1018-0001 8 Ch. Dig. Input 24V, 10µs, M8"}
{attribute addProperty Physics "YY"}
{attribute addProperty Id "Channel_1AT %I*Channel_830843C11Channel_2AT %I*Channel_830843C11Channel_3AT %I*Channel_830843C11Channel_4AT %I*Channel_830843C11Channel_5AT %I*Channel_830843C11Channel_6AT %I*Channel_830843C11Channel_7AT %I*Channel_830843C11Channel_8AT %I*Channel_830843C11WcStateAT %I*WcState_9091E0EB2InfoDataAT %I*InfoData_6F19DB2B2"}
{attribute addProperty CRC "2028524509"}
{attribute addProperty Size "12"}
TYPE EP1018_78E8D3DD EXTENDS EtcSlaveBoxBase_77A0E4A7 :
STRUCT
	{attribute addProperty Name "Channel_1"}
	Channel_1 : Channel_830843C1;
	{attribute addProperty Name "Channel_2"}
	Channel_2 : Channel_830843C1;
	{attribute addProperty Name "Channel_3"}
	Channel_3 : Channel_830843C1;
	{attribute addProperty Name "Channel_4"}
	Channel_4 : Channel_830843C1;
	{attribute addProperty Name "Channel_5"}
	Channel_5 : Channel_830843C1;
	{attribute addProperty Name "Channel_6"}
	Channel_6 : Channel_830843C1;
	{attribute addProperty Name "Channel_7"}
	Channel_7 : Channel_830843C1;
	{attribute addProperty Name "Channel_8"}
	Channel_8 : Channel_830843C1;
	{attribute addProperty Name "WcState"}
	WcState : WcState_9091E0EB;
	{attribute addProperty Name "InfoData"}
	InfoData : InfoData_6F19DB2B;
END_STRUCT
END_TYPE

// ---- DUTs/IO/Boxes/EP1098_78E8D3DD.TcDUT
{attribute 'GeneratedUsingTerminal: EP1098-0001-0016'}
{attribute addProperty BoxType "EP1098-0001-0016"}
{attribute addProperty Description "EP1098-0001 8 Ch. Dig. Input 24V, 10µs, M8, negative"}
{attribute addProperty Physics "YY"}
{attribute addProperty Id "Channel_1AT %I*Channel_830843C11Channel_2AT %I*Channel_830843C11Channel_3AT %I*Channel_830843C11Channel_4AT %I*Channel_830843C11Channel_5AT %I*Channel_830843C11Channel_6AT %I*Channel_830843C11Channel_7AT %I*Channel_830843C11Channel_8AT %I*Channel_830843C11WcStateAT %I*WcState_9091E0EB2InfoDataAT %I*InfoData_6F19DB2B2"}
{attribute addProperty CRC "2028524509"}
{attribute addProperty Size "12"}
TYPE EP1098_78E8D3DD EXTENDS EtcSlaveBoxBase_77A0E4A7 :
STRUCT
	{attribute addProperty Name "Channel_1"}
	Channel_1 : Channel_830843C1;
	{attribute addProperty Name "Channel_2"}
	Channel_2 : Channel_830843C1;
	{attribute addProperty Name "Channel_3"}
	Channel_3 : Channel_830843C1;
	{attribute addProperty Name "Channel_4"}
	Channel_4 : Channel_830843C1;
	{attribute addProperty Name "Channel_5"}
	Channel_5 : Channel_830843C1;
	{attribute addProperty Name "Channel_6"}
	Channel_6 : Channel_830843C1;
	{attribute addProperty Name "Channel_7"}
	Channel_7 : Channel_830843C1;
	{attribute addProperty Name "Channel_8"}
	Channel_8 : Channel_830843C1;
	{attribute addProperty Name "WcState"}
	WcState : WcState_9091E0EB;
	{attribute addProperty Name "InfoData"}
	InfoData : InfoData_6F19DB2B;
END_STRUCT
END_TYPE

// ---- DUTs/IO/Boxes/EP1111_837A6B03.TcDUT
{attribute 'GeneratedUsingTerminal: EP1111-0000-0016'}
{attribute addProperty BoxType "EP1111-0000-0016"}
{attribute addProperty Description "EP1111-0000 ID-Switch"}
{attribute addProperty Physics "YY"}
{attribute addProperty Id "ID_InputsAT %I*ID_Inputs_07C9D28F2WcStateAT %I*WcState_9091E0EB2InfoDataAT %I*InfoData_32EB74EA10"}
{attribute addProperty CRC "2205838083"}
{attribute addProperty Size "14"}
TYPE EP1111_837A6B03 EXTENDS EtcSlaveBoxBase_77A0E4A7 :
STRUCT
	{attribute addProperty Name "ID_Inputs"}
	ID_Inputs : ID_Inputs_07C9D28F;
	{attribute addProperty Name "WcState"}
	WcState : WcState_9091E0EB;
	{attribute addProperty Name "InfoData"}
	InfoData : InfoData_32EB74EA;
END_STRUCT
END_TYPE

// ---- DUTs/IO/Boxes/EP1122_1FC0878B.TcDUT
{attribute 'GeneratedUsingTerminal: EP1122-0001-0016'}
{attribute addProperty BoxType "EP1122-0001-0016"}
{attribute addProperty Description "EP1122-0001 2 port EtherCAT junction"}
{attribute addProperty Physics "YYYY"}
{attribute addProperty Id "InfoDataAT %I*InfoData_6F19DB2B2"}
{attribute addProperty CRC "532711307"}
{attribute addProperty Size "2"}
TYPE EP1122_1FC0878B EXTENDS EtcSlaveBoxBase_77A0E4A7 :
STRUCT
	{attribute addProperty Name "InfoData"}
	InfoData : InfoData_6F19DB2B;
END_STRUCT
END_TYPE

// ---- DUTs/IO/Boxes/EP1258_58F475DD.TcDUT
{attribute 'GeneratedUsingTerminal: EP1258-0001-0016'}
{attribute addProperty BoxType "EP1258-0001-0016"}
{attribute addProperty Description "EP1258-0001 8 Ch. Dig. Input 24V, 10µs, DC Latch, M8"}
{attribute addProperty Physics "YY"}
{attribute addProperty Id "Channel_1AT %I*Channel_830843C11Channel_2AT %I*Channel_830843C11Channel_3AT %I*Channel_830843C11Channel_4AT %I*Channel_830843C11Channel_5AT %I*Channel_830843C11Channel_6AT %I*Channel_830843C11Channel_7AT %I*Channel_830843C11Channel_8AT %I*Channel_830843C11LatchAT %I*Latch_8E41329534WcStateAT %I*WcState_B516A2644InfoDataAT %I*InfoData_A7436BC610"}
{attribute addProperty CRC "1492415965"}
{attribute addProperty Size "56"}
TYPE EP1258_58F475DD EXTENDS EtcSlaveBoxBase_77A0E4A7 :
STRUCT
	{attribute addProperty Name "Channel_1"}
	Channel_1 : Channel_830843C1;
	{attribute addProperty Name "Channel_2"}
	Channel_2 : Channel_830843C1;
	{attribute addProperty Name "Channel_3"}
	Channel_3 : Channel_830843C1;
	{attribute addProperty Name "Channel_4"}
	Channel_4 : Channel_830843C1;
	{attribute addProperty Name "Channel_5"}
	Channel_5 : Channel_830843C1;
	{attribute addProperty Name "Channel_6"}
	Channel_6 : Channel_830843C1;
	{attribute addProperty Name "Channel_7"}
	Channel_7 : Channel_830843C1;
	{attribute addProperty Name "Channel_8"}
	Channel_8 : Channel_830843C1;
	{attribute addProperty Name "Latch"}
	Latch : Latch_8E413295;
	{attribute addProperty Name "WcState"}
	WcState : WcState_B516A264;
	{attribute addProperty Name "InfoData"}
	InfoData : InfoData_A7436BC6;
END_STRUCT
END_TYPE

// ---- DUTs/IO/Boxes/EP1312_1FC0878B.TcDUT
{attribute 'GeneratedUsingTerminal: EP1312-0001-0016'}
{attribute addProperty BoxType "EP1312-0001-0016"}
{attribute addProperty Description "EP1312-0001 2 port EtherCAT P gateway"}
{attribute addProperty Physics "YYYY"}
{attribute addProperty Id "InfoDataAT %I*InfoData_6F19DB2B2"}
{attribute addProperty CRC "532711307"}
{attribute addProperty Size "2"}
TYPE EP1312_1FC0878B EXTENDS EtcSlaveBoxBase_77A0E4A7 :
STRUCT
	{attribute addProperty Name "InfoData"}
	InfoData : InfoData_6F19DB2B;
END_STRUCT
END_TYPE

// ---- DUTs/IO/Boxes/EP1518_CC442588.TcDUT
{attribute 'GeneratedUsingTerminal: EP1518-0002-0016'}
{attribute addProperty BoxType "EP1518-0002-0016"}
{attribute addProperty Description "EP1518-0002 8 Ch. Dig. multi-function Input 24V"}
{attribute addProperty Physics "YY"}
{attribute addProperty Id "CNT_Input_Channel_1AT %I*CNT_Input_Channel_FF10BD3C11CNT_Input_Channel_2AT %I*CNT_Input_Channel_FF10BD3C11DIG_InputsAT %I*DIG_Inputs_CAFF60048DIG_Inputs_DeviceAT %I*DIG_Inputs_Device_1F4E72EB5CNT_Output_Channel_1AT %Q*CNT_Output_Channel_550BB6DF6CNT_Output_Channel_2AT %Q*CNT_Output_Channel_550BB6DF6WcStateAT %I*WcState_9091E0EB2InfoDataAT %I*InfoData_32EB74EA10"}
{attribute addProperty CRC "3427018120"}
{attribute addProperty Size "59"}
TYPE EP1518_CC442588 EXTENDS EtcSlaveBoxBase_77A0E4A7 :
STRUCT
	{attribute addProperty Name "CNT_Input_Channel_1"}
	CNT_Input_Channel_1 : CNT_Input_Channel_FF10BD3C;
	{attribute addProperty Name "CNT_Input_Channel_2"}
	CNT_Input_Channel_2 : CNT_Input_Channel_FF10BD3C;
	{attribute addProperty Name "DIG_Inputs"}
	DIG_Inputs : DIG_Inputs_CAFF6004;
	{attribute addProperty Name "DIG_Inputs_Device"}
	DIG_Inputs_Device : DIG_Inputs_Device_1F4E72EB;
	{attribute addProperty Name "CNT_Output_Channel_1"}
	CNT_Output_Channel_1 : CNT_Output_Channel_550BB6DF;
	{attribute addProperty Name "CNT_Output_Channel_2"}
	CNT_Output_Channel_2 : CNT_Output_Channel_550BB6DF;
	{attribute addProperty Name "WcState"}
	WcState : WcState_9091E0EB;
	{attribute addProperty Name "InfoData"}
	InfoData : InfoData_32EB74EA;
END_STRUCT
END_TYPE

// ---- DUTs/IO/Boxes/EP1809_32157CFD.TcDUT
{attribute 'GeneratedUsingTerminal: EP1809-0021-0016'}
{attribute addProperty BoxType "EP1809-0021-0016"}
{attribute addProperty Description "EP1809-0021 16 Ch. Dig. Input 24V, 3ms, M8"}
{attribute addProperty Physics "YY"}
{attribute addProperty Id "Channel_1AT %I*Channel_830843C11Channel_2AT %I*Channel_830843C11Channel_3AT %I*Channel_830843C11Channel_4AT %I*Channel_830843C11Channel_5AT %I*Channel_830843C11Channel_6AT %I*Channel_830843C11Channel_7AT %I*Channel_830843C11Channel_8AT %I*Channel_830843C11Channel_9AT %I*Channel_830843C11Channel_10AT %I*Channel_830843C11Channel_11AT %I*Channel_830843C11Channel_12AT %I*Channel_830843C11Channel_13AT %I*Channel_830843C11Channel_14AT %I*Channel_830843C11Channel_15AT %I*Channel_830843C11Channel_16AT %I*Channel_830843C11WcStateAT %I*WcState_9091E0EB2InfoDataAT %I*InfoData_6F19DB2B2"}
{attribute addProperty CRC "840269053"}
{attribute addProperty Size "20"}
TYPE EP1809_32157CFD EXTENDS EtcSlaveBoxBase_77A0E4A7 :
STRUCT
	{attribute addProperty Name "Channel_1"}
	Channel_1 : Channel_830843C1;
	{attribute addProperty Name "Channel_2"}
	Channel_2 : Channel_830843C1;
	{attribute addProperty Name "Channel_3"}
	Channel_3 : Channel_830843C1;
	{attribute addProperty Name "Channel_4"}
	Channel_4 : Channel_830843C1;
	{attribute addProperty Name "Channel_5"}
	Channel_5 : Channel_830843C1;
	{attribute addProperty Name "Channel_6"}
	Channel_6 : Channel_830843C1;
	{attribute addProperty Name "Channel_7"}
	Channel_7 : Channel_830843C1;
	{attribute addProperty Name "Channel_8"}
	Channel_8 : Channel_830843C1;
	{attribute addProperty Name "Channel_9"}
	Channel_9 : Channel_830843C1;
	{attribute addProperty Name "Channel_10"}
	Channel_10 : Channel_830843C1;
	{attribute addProperty Name "Channel_11"}
	Channel_11 : Channel_830843C1;
	{attribute addProperty Name "Channel_12"}
	Channel_12 : Channel_830843C1;
	{attribute addProperty Name "Channel_13"}
	Channel_13 : Channel_830843C1;
	{attribute addProperty Name "Channel_14"}
	Channel_14 : Channel_830843C1;
	{attribute addProperty Name "Channel_15"}
	Channel_15 : Channel_830843C1;
	{attribute addProperty Name "Channel_16"}
	Channel_16 : Channel_830843C1;
	{attribute addProperty Name "WcState"}
	WcState : WcState_9091E0EB;
	{attribute addProperty Name "InfoData"}
	InfoData : InfoData_6F19DB2B;
END_STRUCT
END_TYPE

// ---- DUTs/IO/Boxes/EP1809_AA84A50E.TcDUT
{attribute 'GeneratedUsingTerminal: EP1809-0042-0018'}
{attribute addProperty BoxType "EP1809-0042-0018"}
{attribute addProperty Description "EP1809-0042 16 Ch. Dig. Input, 3ms, 24 V DC, M12"}
{attribute addProperty Physics "YY"}
{attribute addProperty Id "DI_X01_Pin4AT %I*DI_X01_Pin_830843C11DI_X01_Pin2AT %I*DI_X01_Pin_830843C11DI_X02_Pin4AT %I*DI_X02_Pin_830843C11DI_X02_Pin2AT %I*DI_X02_Pin_830843C11DI_X03_Pin4AT %I*DI_X03_Pin_830843C11DI_X03_Pin2AT %I*DI_X03_Pin_830843C11DI_X04_Pin4AT %I*DI_X04_Pin_830843C11DI_X04_Pin2AT %I*DI_X04_Pin_830843C11DI_X05_Pin4AT %I*DI_X05_Pin_830843C11DI_X05_Pin2AT %I*DI_X05_Pin_830843C11DI_X06_Pin4AT %I*DI_X06_Pin_830843C11DI_X06_Pin2AT %I*DI_X06_Pin_830843C11DI_X07_Pin4AT %I*DI_X07_Pin_830843C11DI_X07_Pin2AT %I*DI_X07_Pin_830843C11DI_X08_Pin4AT %I*DI_X08_Pin_830843C11DI_X08_Pin2AT %I*DI_X08_Pin_830843C11WcStateAT %I*WcState_9091E0EB2InfoDataAT %I*InfoData_6F19DB2B2"}
{attribute addProperty CRC "2860819726"}
{attribute addProperty Size "20"}
TYPE EP1809_AA84A50E EXTENDS EtcSlaveBoxBase_77A0E4A7 :
STRUCT
	{attribute addProperty Name "DI_X01_Pin4"}
	DI_X01_Pin4 : DI_X01_Pin_830843C1;
	{attribute addProperty Name "DI_X01_Pin2"}
	DI_X01_Pin2 : DI_X01_Pin_830843C1;
	{attribute addProperty Name "DI_X02_Pin4"}
	DI_X02_Pin4 : DI_X02_Pin_830843C1;
	{attribute addProperty Name "DI_X02_Pin2"}
	DI_X02_Pin2 : DI_X02_Pin_830843C1;
	{attribute addProperty Name "DI_X03_Pin4"}
	DI_X03_Pin4 : DI_X03_Pin_830843C1;
	{attribute addProperty Name "DI_X03_Pin2"}
	DI_X03_Pin2 : DI_X03_Pin_830843C1;
	{attribute addProperty Name "DI_X04_Pin4"}
	DI_X04_Pin4 : DI_X04_Pin_830843C1;
	{attribute addProperty Name "DI_X04_Pin2"}
	DI_X04_Pin2 : DI_X04_Pin_830843C1;
	{attribute addProperty Name "DI_X05_Pin4"}
	DI_X05_Pin4 : DI_X05_Pin_830843C1;
	{attribute addProperty Name "DI_X05_Pin2"}
	DI_X05_Pin2 : DI_X05_Pin_830843C1;
	{attribute addProperty Name "DI_X06_Pin4"}
	DI_X06_Pin4 : DI_X06_Pin_830843C1;
	{attribute addProperty Name "DI_X06_Pin2"}
	DI_X06_Pin2 : DI_X06_Pin_830843C1;
	{attribute addProperty Name "DI_X07_Pin4"}
	DI_X07_Pin4 : DI_X07_Pin_830843C1;
	{attribute addProperty Name "DI_X07_Pin2"}
	DI_X07_Pin2 : DI_X07_Pin_830843C1;
	{attribute addProperty Name "DI_X08_Pin4"}
	DI_X08_Pin4 : DI_X08_Pin_830843C1;
	{attribute addProperty Name "DI_X08_Pin2"}
	DI_X08_Pin2 : DI_X08_Pin_830843C1;
	{attribute addProperty Name "WcState"}
	WcState : WcState_9091E0EB;
	{attribute addProperty Name "InfoData"}
	InfoData : InfoData_6F19DB2B;
END_STRUCT
END_TYPE

// ---- DUTs/IO/Boxes/EP1809_8E14C816.TcDUT
{attribute 'GeneratedUsingTerminal: EP1809-0042-0019'}
{attribute addProperty BoxType "EP1809-0042-0019"}
{attribute addProperty Description "EP1809-0042 16 Ch. Dig. Input, 3ms, 24 V DC, M12"}
{attribute addProperty Physics "YY"}
{attribute addProperty Id "DI_X01_4AT %I*DI_X_830843C11DI_X01_2AT %I*DI_X_830843C11DI_X02_4AT %I*DI_X_830843C11DI_X02_2AT %I*DI_X_830843C11DI_X03_4AT %I*DI_X_830843C11DI_X03_2AT %I*DI_X_830843C11DI_X04_4AT %I*DI_X_830843C11DI_X04_2AT %I*DI_X_830843C11DI_X05_4AT %I*DI_X_830843C11DI_X05_2AT %I*DI_X_830843C11DI_X06_4AT %I*DI_X_830843C11DI_X06_2AT %I*DI_X_830843C11DI_X07_4AT %I*DI_X_830843C11DI_X07_2AT %I*DI_X_830843C11DI_X08_4AT %I*DI_X_830843C11DI_X08_2AT %I*DI_X_830843C11WcStateAT %I*WcState_9091E0EB2InfoDataAT %I*InfoData_6F19DB2B2"}
{attribute addProperty CRC "2383726614"}
{attribute addProperty Size "20"}
TYPE EP1809_8E14C816 EXTENDS EtcSlaveBoxBase_77A0E4A7 :
STRUCT
	{attribute addProperty Name "DI_X01_4"}
	DI_X01_4 : DI_X_830843C1;
	{attribute addProperty Name "DI_X01_2"}
	DI_X01_2 : DI_X_830843C1;
	{attribute addProperty Name "DI_X02_4"}
	DI_X02_4 : DI_X_830843C1;
	{attribute addProperty Name "DI_X02_2"}
	DI_X02_2 : DI_X_830843C1;
	{attribute addProperty Name "DI_X03_4"}
	DI_X03_4 : DI_X_830843C1;
	{attribute addProperty Name "DI_X03_2"}
	DI_X03_2 : DI_X_830843C1;
	{attribute addProperty Name "DI_X04_4"}
	DI_X04_4 : DI_X_830843C1;
	{attribute addProperty Name "DI_X04_2"}
	DI_X04_2 : DI_X_830843C1;
	{attribute addProperty Name "DI_X05_4"}
	DI_X05_4 : DI_X_830843C1;
	{attribute addProperty Name "DI_X05_2"}
	DI_X05_2 : DI_X_830843C1;
	{attribute addProperty Name "DI_X06_4"}
	DI_X06_4 : DI_X_830843C1;
	{attribute addProperty Name "DI_X06_2"}
	DI_X06_2 : DI_X_830843C1;
	{attribute addProperty Name "DI_X07_4"}
	DI_X07_4 : DI_X_830843C1;
	{attribute addProperty Name "DI_X07_2"}
	DI_X07_2 : DI_X_830843C1;
	{attribute addProperty Name "DI_X08_4"}
	DI_X08_4 : DI_X_830843C1;
	{attribute addProperty Name "DI_X08_2"}
	DI_X08_2 : DI_X_830843C1;
	{attribute addProperty Name "WcState"}
	WcState : WcState_9091E0EB;
	{attribute addProperty Name "InfoData"}
	InfoData : InfoData_6F19DB2B;
END_STRUCT
END_TYPE

// ---- DUTs/IO/Boxes/EP1816_73178B54.TcDUT
{attribute 'GeneratedUsingTerminal: EP1816-0003-0016'}
{attribute addProperty BoxType "EP1816-0003-0016"}
{attribute addProperty Description "EP1816-0003 16 Ch. Dig. Input 24V, 10µs, 10-Pole Plug Connector"}
{attribute addProperty Physics "YY"}
{attribute addProperty Id "DIG_Inputs_Channel_1AT %I*DIG_Inputs_Channel_ACAA042510DIG_Inputs_Channel_2AT %I*DIG_Inputs_Channel_ACAA042510WcStateAT %I*WcState_9091E0EB2InfoDataAT %I*InfoData_32EB74EA10"}
{attribute addProperty CRC "1930922836"}
{attribute addProperty Size "32"}
TYPE EP1816_73178B54 EXTENDS EtcSlaveBoxBase_77A0E4A7 :
STRUCT
	{attribute addProperty Name "DIG_Inputs_Channel_1"}
	DIG_Inputs_Channel_1 : DIG_Inputs_Channel_ACAA0425;
	{attribute addProperty Name "DIG_Inputs_Channel_2"}
	DIG_Inputs_Channel_2 : DIG_Inputs_Channel_ACAA0425;
	{attribute addProperty Name "WcState"}
	WcState : WcState_9091E0EB;
	{attribute addProperty Name "InfoData"}
	InfoData : InfoData_32EB74EA;
END_STRUCT
END_TYPE

// ---- DUTs/IO/Boxes/EP1816_03D88109.TcDUT
{attribute 'GeneratedUsingTerminal: EP1816-0008-0016'}
{attribute addProperty BoxType "EP1816-0008-0016"}
{attribute addProperty Description "EP1816-0008 16 Ch. Dig. Input 24V, 10µs, D-SUB25"}
{attribute addProperty Physics "YY"}
{attribute addProperty Id "DO_Inputs_Channel_1AT %I*DO_Inputs_Channel_CC4551489DO_Inputs_Channel_2AT %I*DO_Inputs_Channel_CC4551489WcStateAT %I*WcState_9091E0EB2InfoDataAT %I*InfoData_32EB74EA10"}
{attribute addProperty CRC "64520457"}
{attribute addProperty Size "30"}
TYPE EP1816_03D88109 EXTENDS EtcSlaveBoxBase_77A0E4A7 :
STRUCT
	{attribute addProperty Name "DO_Inputs_Channel_1"}
	DO_Inputs_Channel_1 : DO_Inputs_Channel_CC455148;
	{attribute addProperty Name "DO_Inputs_Channel_2"}
	DO_Inputs_Channel_2 : DO_Inputs_Channel_CC455148;
	{attribute addProperty Name "WcState"}
	WcState : WcState_9091E0EB;
	{attribute addProperty Name "InfoData"}
	InfoData : InfoData_32EB74EA;
END_STRUCT
END_TYPE

// ---- DUTs/IO/Boxes/EP1816_5E50D3DD.TcDUT
{attribute 'GeneratedUsingTerminal: EP1816-0008-0018'}
{attribute addProperty BoxType "EP1816-0008-0018"}
{attribute addProperty Description "EP1816-0008 16 Ch. Dig. Input 24V, 10µs, D-SUB25"}
{attribute addProperty Physics "YY"}
{attribute addProperty Id "DIG_Inputs_Channel_1AT %I*DIG_Inputs_Channel_CC4551489DIG_Inputs_Channel_2AT %I*DIG_Inputs_Channel_CC4551489WcStateAT %I*WcState_9091E0EB2InfoDataAT %I*InfoData_32EB74EA10"}
{attribute addProperty CRC "1582355421"}
{attribute addProperty Size "30"}
TYPE EP1816_5E50D3DD EXTENDS EtcSlaveBoxBase_77A0E4A7 :
STRUCT
	{attribute addProperty Name "DIG_Inputs_Channel_1"}
	DIG_Inputs_Channel_1 : DIG_Inputs_Channel_CC455148;
	{attribute addProperty Name "DIG_Inputs_Channel_2"}
	DIG_Inputs_Channel_2 : DIG_Inputs_Channel_CC455148;
	{attribute addProperty Name "WcState"}
	WcState : WcState_9091E0EB;
	{attribute addProperty Name "InfoData"}
	InfoData : InfoData_32EB74EA;
END_STRUCT
END_TYPE

// ---- DUTs/IO/Boxes/EP1816_F50297FE.TcDUT
{attribute 'GeneratedUsingTerminal: EP1816-1008-0016'}
{attribute addProperty BoxType "EP1816-1008-0016"}
{attribute addProperty Description "EP1816-1008 16Ch. Dig. Input  24V 10µs, DSUB-25"}
{attribute addProperty Physics "YY"}
{attribute addProperty Id "DIG_Inputs_Channel_1AT %I*DIG_Inputs_Channel_38F9DD278DIG_Inputs_Channel_2AT %I*DIG_Inputs_Channel_38F9DD278DIG_Inputs_DeviceAT %I*DIG_Inputs_Device_B3EA42044WcStateAT %I*WcState_9091E0EB2InfoDataAT %I*InfoData_32EB74EA10"}
{attribute addProperty CRC "4110587902"}
{attribute addProperty Size "32"}
TYPE EP1816_F50297FE EXTENDS EtcSlaveBoxBase_77A0E4A7 :
STRUCT
	{attribute addProperty Name "DIG_Inputs_Channel_1"}
	DIG_Inputs_Channel_1 : DIG_Inputs_Channel_38F9DD27;
	{attribute addProperty Name "DIG_Inputs_Channel_2"}
	DIG_Inputs_Channel_2 : DIG_Inputs_Channel_38F9DD27;
	{attribute addProperty Name "DIG_Inputs_Device"}
	DIG_Inputs_Device : DIG_Inputs_Device_B3EA4204;
	{attribute addProperty Name "WcState"}
	WcState : WcState_9091E0EB;
	{attribute addProperty Name "InfoData"}
	InfoData : InfoData_32EB74EA;
END_STRUCT
END_TYPE

// ---- DUTs/IO/Boxes/EP1816_CABD51E6.TcDUT
{attribute 'GeneratedUsingTerminal: EP1816-3008-0016'}
{attribute addProperty BoxType "EP1816-3008-0016"}
{attribute addProperty Description "EP1816-3008 16Ch. Dig. Input  24V 10µs Acceleration Sensor, DSUB-25"}
{attribute addProperty Physics "YY"}
{attribute addProperty Id "DIG_Inputs_Channel_1AT %I*DIG_Inputs_Channel_38F9DD278DIG_Inputs_Channel_2AT %I*DIG_Inputs_Channel_38F9DD278AI_Inputs_Channel_1AT %I*AI_Inputs_Channel_C3DE7A0A4AI_Inputs_Channel_2AT %I*AI_Inputs_Channel_C3DE7A0A4AI_Inputs_Channel_3AT %I*AI_Inputs_Channel_C3DE7A0A4AI_Inputs_Channel_4AT %I*AI_Inputs_Channel_C3DE7A0A4AI_Inputs_Channel_5AT %I*AI_Inputs_Channel_C3DE7A0A4AI_Inputs_Channel_6AT %I*AI_Inputs_Channel_C3DE7A0A4DIG_Inputs_DeviceAT %I*DIG_Inputs_Device_B3EA42044WcStateAT %I*WcState_9091E0EB2InfoDataAT %I*InfoData_32EB74EA10"}
{attribute addProperty CRC "3401404902"}
{attribute addProperty Size "56"}
TYPE EP1816_CABD51E6 EXTENDS EtcSlaveBoxBase_77A0E4A7 :
STRUCT
	{attribute addProperty Name "DIG_Inputs_Channel_1"}
	DIG_Inputs_Channel_1 : DIG_Inputs_Channel_38F9DD27;
	{attribute addProperty Name "DIG_Inputs_Channel_2"}
	DIG_Inputs_Channel_2 : DIG_Inputs_Channel_38F9DD27;
	{attribute addProperty Name "AI_Inputs_Channel_1"}
	AI_Inputs_Channel_1 : AI_Inputs_Channel_C3DE7A0A;
	{attribute addProperty Name "AI_Inputs_Channel_2"}
	AI_Inputs_Channel_2 : AI_Inputs_Channel_C3DE7A0A;
	{attribute addProperty Name "AI_Inputs_Channel_3"}
	AI_Inputs_Channel_3 : AI_Inputs_Channel_C3DE7A0A;
	{attribute addProperty Name "AI_Inputs_Channel_4"}
	AI_Inputs_Channel_4 : AI_Inputs_Channel_C3DE7A0A;
	{attribute addProperty Name "AI_Inputs_Channel_5"}
	AI_Inputs_Channel_5 : AI_Inputs_Channel_C3DE7A0A;
	{attribute addProperty Name "AI_Inputs_Channel_6"}
	AI_Inputs_Channel_6 : AI_Inputs_Channel_C3DE7A0A;
	{attribute addProperty Name "DIG_Inputs_Device"}
	DIG_Inputs_Device : DIG_Inputs_Device_B3EA4204;
	{attribute addProperty Name "WcState"}
	WcState : WcState_9091E0EB;
	{attribute addProperty Name "InfoData"}
	InfoData : InfoData_32EB74EA;
END_STRUCT
END_TYPE

// ---- DUTs/IO/Boxes/EP1819_32157CFD.TcDUT
{attribute 'GeneratedUsingTerminal: EP1819-0021-0016'}
{attribute addProperty BoxType "EP1819-0021-0016"}
{attribute addProperty Description "EP1819-0021 16 Ch. Dig. Input 24V, 10µs, M8"}
{attribute addProperty Physics "YY"}
{attribute addProperty Id "Channel_1AT %I*Channel_830843C11Channel_2AT %I*Channel_830843C11Channel_3AT %I*Channel_830843C11Channel_4AT %I*Channel_830843C11Channel_5AT %I*Channel_830843C11Channel_6AT %I*Channel_830843C11Channel_7AT %I*Channel_830843C11Channel_8AT %I*Channel_830843C11Channel_9AT %I*Channel_830843C11Channel_10AT %I*Channel_830843C11Channel_11AT %I*Channel_830843C11Channel_12AT %I*Channel_830843C11Channel_13AT %I*Channel_830843C11Channel_14AT %I*Channel_830843C11Channel_15AT %I*Channel_830843C11Channel_16AT %I*Channel_830843C11WcStateAT %I*WcState_9091E0EB2InfoDataAT %I*InfoData_6F19DB2B2"}
{attribute addProperty CRC "840269053"}
{attribute addProperty Size "20"}
TYPE EP1819_32157CFD EXTENDS EtcSlaveBoxBase_77A0E4A7 :
STRUCT
	{attribute addProperty Name "Channel_1"}
	Channel_1 : Channel_830843C1;
	{attribute addProperty Name "Channel_2"}
	Channel_2 : Channel_830843C1;
	{attribute addProperty Name "Channel_3"}
	Channel_3 : Channel_830843C1;
	{attribute addProperty Name "Channel_4"}
	Channel_4 : Channel_830843C1;
	{attribute addProperty Name "Channel_5"}
	Channel_5 : Channel_830843C1;
	{attribute addProperty Name "Channel_6"}
	Channel_6 : Channel_830843C1;
	{attribute addProperty Name "Channel_7"}
	Channel_7 : Channel_830843C1;
	{attribute addProperty Name "Channel_8"}
	Channel_8 : Channel_830843C1;
	{attribute addProperty Name "Channel_9"}
	Channel_9 : Channel_830843C1;
	{attribute addProperty Name "Channel_10"}
	Channel_10 : Channel_830843C1;
	{attribute addProperty Name "Channel_11"}
	Channel_11 : Channel_830843C1;
	{attribute addProperty Name "Channel_12"}
	Channel_12 : Channel_830843C1;
	{attribute addProperty Name "Channel_13"}
	Channel_13 : Channel_830843C1;
	{attribute addProperty Name "Channel_14"}
	Channel_14 : Channel_830843C1;
	{attribute addProperty Name "Channel_15"}
	Channel_15 : Channel_830843C1;
	{attribute addProperty Name "Channel_16"}
	Channel_16 : Channel_830843C1;
	{attribute addProperty Name "WcState"}
	WcState : WcState_9091E0EB;
	{attribute addProperty Name "InfoData"}
	InfoData : InfoData_6F19DB2B;
END_STRUCT
END_TYPE

// ---- DUTs/IO/Boxes/EP1859_B704EC1A.TcDUT
{attribute 'GeneratedUsingTerminal: EP1859-0042-0018'}
{attribute addProperty BoxType "EP1859-0042-0018"}
{attribute addProperty Description "EP1859-0042 8 Ch. Dig. In, 3ms, 8 Ch. Dig. Out 24V, 0.5A, M12 "}
{attribute addProperty Physics "YY"}
{attribute addProperty Id "DI_X01_Pin4AT %I*DI_X01_Pin_830843C11DI_X01_Pin2AT %I*DI_X01_Pin_830843C11DI_X02_Pin4AT %I*DI_X02_Pin_830843C11DI_X02_Pin2AT %I*DI_X02_Pin_830843C11DI_X03_Pin4AT %I*DI_X03_Pin_830843C11DI_X03_Pin2AT %I*DI_X03_Pin_830843C11DI_X04_Pin4AT %I*DI_X04_Pin_830843C11DI_X04_Pin2AT %I*DI_X04_Pin_830843C11DO_X05_Pin4AT %Q*DO_X05_Pin_42CA91F71DO_X05_Pin2AT %Q*DO_X05_Pin_42CA91F71DO_X06_Pin4AT %Q*DO_X06_Pin_42CA91F71DO_X06_Pin2AT %Q*DO_X06_Pin_42CA91F71DO_X07_Pin4AT %Q*DO_X07_Pin_42CA91F71DO_X07_Pin2AT %Q*DO_X07_Pin_42CA91F71DO_X08_Pin4AT %Q*DO_X08_Pin_42CA91F71DO_X08_Pin2AT %Q*DO_X08_Pin_42CA91F71WcStateAT %I*WcState_9091E0EB2InfoDataAT %I*InfoData_6F19DB2B2"}
{attribute addProperty CRC "3070553114"}
{attribute addProperty Size "20"}
TYPE EP1859_B704EC1A EXTENDS EtcSlaveBoxBase_77A0E4A7 :
STRUCT
	{attribute addProperty Name "DI_X01_Pin4"}
	DI_X01_Pin4 : DI_X01_Pin_830843C1;
	{attribute addProperty Name "DI_X01_Pin2"}
	DI_X01_Pin2 : DI_X01_Pin_830843C1;
	{attribute addProperty Name "DI_X02_Pin4"}
	DI_X02_Pin4 : DI_X02_Pin_830843C1;
	{attribute addProperty Name "DI_X02_Pin2"}
	DI_X02_Pin2 : DI_X02_Pin_830843C1;
	{attribute addProperty Name "DI_X03_Pin4"}
	DI_X03_Pin4 : DI_X03_Pin_830843C1;
	{attribute addProperty Name "DI_X03_Pin2"}
	DI_X03_Pin2 : DI_X03_Pin_830843C1;
	{attribute addProperty Name "DI_X04_Pin4"}
	DI_X04_Pin4 : DI_X04_Pin_830843C1;
	{attribute addProperty Name "DI_X04_Pin2"}
	DI_X04_Pin2 : DI_X04_Pin_830843C1;
	{attribute addProperty Name "DO_X05_Pin4"}
	DO_X05_Pin4 : DO_X05_Pin_42CA91F7;
	{attribute addProperty Name "DO_X05_Pin2"}
	DO_X05_Pin2 : DO_X05_Pin_42CA91F7;
	{attribute addProperty Name "DO_X06_Pin4"}
	DO_X06_Pin4 : DO_X06_Pin_42CA91F7;
	{attribute addProperty Name "DO_X06_Pin2"}
	DO_X06_Pin2 : DO_X06_Pin_42CA91F7;
	{attribute addProperty Name "DO_X07_Pin4"}
	DO_X07_Pin4 : DO_X07_Pin_42CA91F7;
	{attribute addProperty Name "DO_X07_Pin2"}
	DO_X07_Pin2 : DO_X07_Pin_42CA91F7;
	{attribute addProperty Name "DO_X08_Pin4"}
	DO_X08_Pin4 : DO_X08_Pin_42CA91F7;
	{attribute addProperty Name "DO_X08_Pin2"}
	DO_X08_Pin2 : DO_X08_Pin_42CA91F7;
	{attribute addProperty Name "WcState"}
	WcState : WcState_9091E0EB;
	{attribute addProperty Name "InfoData"}
	InfoData : InfoData_6F19DB2B;
END_STRUCT
END_TYPE

// ---- DUTs/IO/Boxes/EP1859_B9D5A785.TcDUT
{attribute 'GeneratedUsingTerminal: EP1859-0042-0019'}
{attribute addProperty BoxType "EP1859-0042-0019"}
{attribute addProperty Description "EP1859-0042 8 Ch. Dig. In, 3ms, 8 Ch. Dig. Out 24V, 0.5A, M12 "}
{attribute addProperty Physics "YY"}
{attribute addProperty Id "DI_X01_4AT %I*DI_X_830843C11DI_X01_2AT %I*DI_X_830843C11DI_X02_4AT %I*DI_X_830843C11DI_X02_2AT %I*DI_X_830843C11DI_X03_4AT %I*DI_X_830843C11DI_X03_2AT %I*DI_X_830843C11DI_X04_4AT %I*DI_X_830843C11DI_X04_2AT %I*DI_X_830843C11DO_X05_4AT %Q*DO_X_42CA91F71DO_X05_2AT %Q*DO_X_42CA91F71DO_X06_4AT %Q*DO_X_42CA91F71DO_X06_2AT %Q*DO_X_42CA91F71DO_X07_4AT %Q*DO_X_42CA91F71DO_X07_2AT %Q*DO_X_42CA91F71DO_X08_4AT %Q*DO_X_42CA91F71DO_X08_2AT %Q*DO_X_42CA91F71WcStateAT %I*WcState_9091E0EB2InfoDataAT %I*InfoData_6F19DB2B2"}
{attribute addProperty CRC "3117787013"}
{attribute addProperty Size "20"}
TYPE EP1859_B9D5A785 EXTENDS EtcSlaveBoxBase_77A0E4A7 :
STRUCT
	{attribute addProperty Name "DI_X01_4"}
	DI_X01_4 : DI_X_830843C1;
	{attribute addProperty Name "DI_X01_2"}
	DI_X01_2 : DI_X_830843C1;
	{attribute addProperty Name "DI_X02_4"}
	DI_X02_4 : DI_X_830843C1;
	{attribute addProperty Name "DI_X02_2"}
	DI_X02_2 : DI_X_830843C1;
	{attribute addProperty Name "DI_X03_4"}
	DI_X03_4 : DI_X_830843C1;
	{attribute addProperty Name "DI_X03_2"}
	DI_X03_2 : DI_X_830843C1;
	{attribute addProperty Name "DI_X04_4"}
	DI_X04_4 : DI_X_830843C1;
	{attribute addProperty Name "DI_X04_2"}
	DI_X04_2 : DI_X_830843C1;
	{attribute addProperty Name "DO_X05_4"}
	DO_X05_4 : DO_X_42CA91F7;
	{attribute addProperty Name "DO_X05_2"}
	DO_X05_2 : DO_X_42CA91F7;
	{attribute addProperty Name "DO_X06_4"}
	DO_X06_4 : DO_X_42CA91F7;
	{attribute addProperty Name "DO_X06_2"}
	DO_X06_2 : DO_X_42CA91F7;
	{attribute addProperty Name "DO_X07_4"}
	DO_X07_4 : DO_X_42CA91F7;
	{attribute addProperty Name "DO_X07_2"}
	DO_X07_2 : DO_X_42CA91F7;
	{attribute addProperty Name "DO_X08_4"}
	DO_X08_4 : DO_X_42CA91F7;
	{attribute addProperty Name "DO_X08_2"}
	DO_X08_2 : DO_X_42CA91F7;
	{attribute addProperty Name "WcState"}
	WcState : WcState_9091E0EB;
	{attribute addProperty Name "InfoData"}
	InfoData : InfoData_6F19DB2B;
END_STRUCT
END_TYPE

// ---- DUTs/IO/Boxes/EP2001_C23D36A6.TcDUT
{attribute 'GeneratedUsingTerminal: EP2001-1000-0016'}
{attribute addProperty BoxType "EP2001-1000-0016"}
{attribute addProperty Description "EP2001-1000 8 Ch. Dig. Output 24V, 0,5A, M8"}
{attribute addProperty Physics "YY"}
{attribute addProperty Id "Group_0AT %Q*Group_99EF3D304Group_1AT %Q*Group_8FCDB3954WcStateAT %I*WcState_0B2B16F91InfoDataAT %I*InfoData_6F19DB2B2"}
{attribute addProperty CRC "3258791590"}
{attribute addProperty Size "11"}
TYPE EP2001_C23D36A6 EXTENDS EtcSlaveBoxBase_77A0E4A7 :
STRUCT
	{attribute addProperty Name "Group_0"}
	Group_0 : Group_99EF3D30;
	{attribute addProperty Name "Group_1"}
	Group_1 : Group_8FCDB395;
	{attribute addProperty Name "WcState"}
	WcState : WcState_0B2B16F9;
	{attribute addProperty Name "InfoData"}
	InfoData : InfoData_6F19DB2B;
END_STRUCT
END_TYPE

